				(* Se non ho abilitato il tasteggio in fase di deposito pacco orrizzontale e la missione non prevede deposito orrizzintale do la quota reale*)
				IF TFProgramma_Ciclo_Lastra.DisabilitaDepositoConTasteggio THEN
					TFProgramma_Ciclo_Lastra.Quota_StartLenta_Deposito_Lastra_Z			:= Traiettoria^.PuntoDiApproccioEndPoint.Z;
					TFProgramma_Ciclo_Lastra.Quota_Deposito_Lastra_Z						:= Traiettoria^.EndPoint.Z;
				ELSE // Altrimenti faccio scendere di più l'asse Z in modo da far avvenire il tasteggio.....
					TFProgramma_Ciclo_Lastra.Quota_StartLenta_Deposito_Lastra_Z			:= Traiettoria^.PuntoDiApproccioEndPoint.Z + 10;
					TFProgramma_Ciclo_Lastra.Quota_Deposito_Lastra_Z						:= Traiettoria^.EndPoint.Z - 100;
				END_IF
				
				TFProgramma_Ciclo_Lastra.Quota_Fuori_Ingombro_ConCarico_Z		:= QuotaFuoriIngombro_Z_ConPEZZO;
				TFProgramma_Ciclo_Lastra.Quota_Fuori_Ingombro_SenzaCarico_Z	:= QuotaFuoriIngombro_Z_AVUOTO;
				
				(*J*)
				TFProgramma_Ciclo_Lastra.Quota_Rotazione_Prelievo_Lastra 			:= Traiettoria^.StartPoint.J;
				TFProgramma_Ciclo_Lastra.Quota_Rotazione_Deposito_Lastra 			:= Traiettoria^.EndPoint.J;
				TFProgramma_Ciclo_Lastra();
				IF TFProgramma_Ciclo_Lastra.Inizializzato THEN
					(* Valuto se è abilitata l'interpolazione degli assi *)
					IF NOT AbilitaInterpolazioneAssi^ THEN
						TFWorkFlowCase(ADR(WorkFlow[NumeroWF]),20,WorkflowCase_JMP);	// Case con FB SENZA interpolazione
					ELSE
						TFWorkFlowCase(ADR(WorkFlow[NumeroWF]),30,WorkflowCase_JMP);	// Case con FB CON interpolazione
					END_IF
				END_IF
				
				PaccoPresoXDataLogger := TRUE;
			END_IF;
		(* Case 20 - Chiamata FB del ciclo di lavoro SENZA INTERPOLAZIONE ASSI *)	
		20:	
			TFWorkFlowCase(ADR(WorkFlow[NumeroWF]),30,WorkflowCase_JMP);	// Case con FB CON interpolazione

		
		(* Case 30 - Chiamata FB del ciclo di lavoro CON INTERPOLAZIONE ASSI *)	
		30:	
			IF CmdExe.RapidStopRequest > 0 OR
				TFPalletizerIsModuleError(Modules) THEN
				TFCiclo_Deposito_Lastra.InterrompiCiclo := TRUE;
			ELSE
				TFCiclo_Deposito_Lastra.InterrompiCiclo := FALSE;
			END_IF
			TFCiclo_Deposito_Lastra.Ciclo					:= ADR(Ciclo_Deposito_Lastra);
			TFCiclo_Deposito_Lastra.Programma				:= ADR(TFProgramma_Ciclo_Lastra);
			TFCiclo_Deposito_Lastra.ModuleAX_X 				:= ADR(Modules^.AX_X);
			TFCiclo_Deposito_Lastra.ModuleAX_Y 				:= ADR(Modules^.AX_Y);
			TFCiclo_Deposito_Lastra.ModuleAX_Z 				:= ADR(Modules^.AX_Z);
			TFCiclo_Deposito_Lastra.ModuleAX_J 				:= ADR(Modules^.AX_J);
			TFCiclo_Deposito_Lastra.ModulePinza 		:= ADR(Modules^.Pinza);
			TFCiclo_Deposito_Lastra.StartInterpolazioneAssi 				:= ADR(STARTInterpolazioneASSI^);
			TFCiclo_Deposito_Lastra.AbilitazioneAnticipoDinamicoMovimenti 	:= AbilitaAnticipoDinamico^;
			//TFCiclo_Deposito_Lastra.AbilitaDepositoPaccoOrrizzontaleConTasteggio	:= (AbilitaDepositoPaccoOrrizzonataleConTasteggio^ AND NOT SimulazioneSenzaPalletFalde);
			//TFCiclo_Deposito_Lastra.AbilitaAccostamentoAsseZ						:= AbilitaAccostamentoAsseZ^;
			TFCiclo_Deposito_Lastra.AbilitazioneGlobalePassMode 					:= Traiettoria^.PassModeGlobalEnable;
			TFCiclo_Deposito_Lastra.Abilita_Ciclo_Step								:= AbilitazioCiclo_TEST_STEP;
			
			IF CommandSTEP AND NOT CommandSTEPTRIG THEN
				TFCiclo_Deposito_Lastra.Command_Step	:= TRUE;
				CommandSTEPTRIG := TRUE;
			ELSIF NOT CommandSTEP AND NOT CommandSTEPTRIG THEN
				TFCiclo_Deposito_Lastra.Command_Step	:= FALSE;
				CommandSTEPTRIG := FALSE;
				CommandSTEP := FALSE;
			ELSIF  STEPCicloDONE THEN
				TFCiclo_Deposito_Lastra.Command_Step	:= FALSE;
				CommandSTEP := FALSE;
				CommandSTEPTRIG := FALSE;
			END_IF
			
			TFCiclo_Deposito_Lastra();
			STEPCicloDONE := TFCiclo_Deposito_Lastra.STEPDone;
			
			IF Ciclo_Deposito_Lastra.Stato = TERMINATO THEN
				OUT.StartTilter := TRUE;
				ProductOnGripper := KNOPRODUCT;
				TFWorkFlowCase(ADR(WorkFlow[NumeroWF]),100,WorkflowCase_JMP);
			ELSIF Ciclo_Deposito_Lastra.Stato = INTERROTTO THEN	
				TFWorkFlowCase(ADR(WorkFlow[NumeroWF]),999,WorkflowCase_JMP);	
					
			END_IF

		(* Case 100 *)
		100:WorkFlow[NumeroWF].State := StateWF_END;
			WorkFlow[NumeroWF].Enable := FALSE;
			CommandSTEP := FALSE;
			CommandSTEPTRIG := FALSE;
			ResetComandoRibaltinoEseguito := FALSE;
			AssiInterpolati := FALSE;

		(* Case 999 *)
		(* WorkFlow ERROR *)
		StateWF_ERROR:
			TFWorkFlowError(ADR(WorkFlow[NumeroWF]),ADR(WorkFlowErrorLog[NumeroWF]));
			CmdExe.PhaseStopRequest := 1;
			CmdExe.RapidStopRequest := 1;
			WorkFlow[NumeroWF].Enable := FALSE;
			CommandSTEP := FALSE;
			CommandSTEPTRIG := FALSE;
			AssiInterpolati := FALSE;
		
		ELSE						
			TFWorkFlowError(ADR(WorkFlow[NumeroWF]),ADR(WorkFlowErrorLog[NumeroWF]));
			TFError(ErrNOCMDCASE,ErrNULL,ADR(CmdExe),ADR(State),ADR(Error),ADR(ErrorLog));	
	END_CASE;
END_IF
END_ACTION

ACTION WF09_CicloDepLastraDaWA:
(*-------------------------------------------------------------------------------------------*)
(* WorkFlow 9 -  CICLO DEPOSITO LASTRA PP *)
(*-------------------------------------------------------------------------------------------*)	
NumeroWF := 9;	
IF WorkFlow[NumeroWF].Enable THEN

	IF NOT TFCommandCaseIsEnable(ADR(CmdExe)) THEN RETURN; END_IF
	CASE WorkFlow[NumeroWF].WFCase OF

		(* Case 0 *)
		0:  WorkFlow[NumeroWF].State := StateWF_RUN;
			STEPCicloDONE := FALSE;	
			TFWorkFlowCase(ADR(WorkFlow[NumeroWF]),1,WorkflowCase_INC);
	
		(* Case 1 - Chiamata del FB del ciclo di riposo per Valorizzarne i valori*)
		1:	IF CmdExe.RapidStopRequest > 0  OR
				TFPalletizerIsModuleError(Modules) THEN
				TFWorkFlowCase(ADR(WorkFlow[NumeroWF]),100,WorkflowCase_JMP);
			ELSE

				TFProgramma_Ciclo_Lastra.X_Par := ParametriProgramma_X_CicloLastra;
				TFProgramma_Ciclo_Lastra.Y_Par := ParametriProgramma_Y_CicloLastra;
				TFProgramma_Ciclo_Lastra.Z_Par := ParametriProgramma_Z_CicloLastra;
				TFProgramma_Ciclo_Lastra.J_Par := ParametriProgramma_J_CicloLastra;
				
				(*X*)
				TFProgramma_Ciclo_Lastra.Quota_StartLenta_Prelievo_Lastra_X			:= Traiettoria^.PuntoDiApproccioStartPoint.X;
				TFProgramma_Ciclo_Lastra.Quota_Prelievo_Lastra_X 					:= Traiettoria^.StartPoint.X;
				TFProgramma_Ciclo_Lastra.Quota_StartLenta_Deposito_Lastra_X	 		:= Traiettoria^.PuntoDiApproccioEndPoint.X;	
				TFProgramma_Ciclo_Lastra.Quota_Deposito_Lastra_X 					:= Traiettoria^.EndPoint.X;
				TFProgramma_Ciclo_Lastra.Quota_Fuori_Ingombro_SenzaCarico_X			:= Traiettoria^.EndPoint.X;
				TFProgramma_Ciclo_Lastra.Quota_Fuori_Ingombro_Carico_X				:= Traiettoria^.EndPoint.X;
				
				//*************************
			   	CoordenadaPosGiroPieza_X 											:= WorkArea^[NuPosGuiroPiking].X ;
				TFProgramma_Ciclo_Lastra.Quota_PosGiroPiezaTraCavalleteX			:= CoordenadaPosGiroPieza_X ;
				//*****************************
				
				(*Y*)
				TFProgramma_Ciclo_Lastra.Quota_StartLenta_Prelievo_Lastra_Y         := Traiettoria^.PuntoDiApproccioStartPoint.Y;;
				TFProgramma_Ciclo_Lastra.Quota_Prelievo_Lastra_Y 					:= Traiettoria^.StartPoint.Y;
				TFProgramma_Ciclo_Lastra.Quota_Distacco_Lastra_Y					:= Traiettoria^.PuntoDiPostPosizionamentoStartPoint.Y;
				TFProgramma_Ciclo_Lastra.Quota_StartLenta_Deposito_Lastra_Y			:= Traiettoria^.PuntoDiApproccioEndPoint.Y;
				TFProgramma_Ciclo_Lastra.Quota_Deposito_Lastra_Y 					:= Traiettoria^.EndPoint.Y;
				TFProgramma_Ciclo_Lastra.Quota_Fuori_Ingombro_Y 					:= QuotaFuoriIngombro_Y_ConCARICO;//DEVE ESSERE GUALE A QUELLE DEL CORRIDOIO
				TFProgramma_Ciclo_Lastra.Quota_PasilloCavallete0GradosY             := CoordenadaPasillo0_Y ;
				TFProgramma_Ciclo_Lastra.Quota_PasilloCavallete1800GradosY          := CoordenadaPasillo180_Y ;
			
				(*Z*)
				TFProgramma_Ciclo_Lastra.Quota_StartLenta_Prelievo_Lastra_Z 		:= MAX(Traiettoria^.PuntoDiApproccioStartPoint.Z,AxisPar_Z.MinPosition+1);
				TFProgramma_Ciclo_Lastra.Quota_Prelievo_Lastra_Z 					:= MAX(Traiettoria^.StartPoint.Z,AxisPar_Z.MinPosition+1);
				TFProgramma_Ciclo_Lastra.Quota_StartLenta_Deposito_Lastra_Z			:= Traiettoria^.PuntoDiApproccioEndPoint.Z;
				TFProgramma_Ciclo_Lastra.Quota_Deposito_Lastra_Z					:= MAX(Traiettoria^.EndPoint.Z,AxisPar_Z.MinPosition+1);
				TFProgramma_Ciclo_Lastra.Quota_Fuori_Ingombro_ConCarico_Z			:= QuotaFuoriIngombro_Z_ConPEZZO;
				TFProgramma_Ciclo_Lastra.Quota_Fuori_Ingombro_SenzaCarico_Z			:= QuotaFuoriIngombro_Z_AVUOTO;
				TFProgramma_Ciclo_Lastra.Quota_Distacco_Lastra_Z					:= Traiettoria^.PuntoDiPostPosizionamentoStartPoint.Z;
				TFProgramma_Ciclo_Lastra.Quota_PostScarico							:= Z_Riposo;	
			
				(*J*)
				TFProgramma_Ciclo_Lastra.Quota_Rotazione_Prelievo_Lastra 			:= Traiettoria^.StartPoint.J;
				TFProgramma_Ciclo_Lastra.Quota_Rotazione_Deposito_Lastra 			:= Traiettoria^.EndPoint.J;
				TFProgramma_Ciclo_Lastra.Quota_Rotazione_StartTasteggio_Lastra		:= Traiettoria^.PuntoDiApproccioStartPoint.J;
				TFProgramma_Ciclo_Lastra.Quota_Fuori_Ingombro_J						:= QuotaFuoriIngombro_J_ConCARICO;
				TFProgramma_Ciclo_Lastra.Quota_Rotazione_Sfogliatura 				:= Traiettoria^.StartPoint.J + HMI_GradiSfogliaturaJ;
				TFProgramma_Ciclo_Lastra.Quota_Posicion_Giro_Pinza					:= WorkSpace^.Y / 2 +900;
				TFProgramma_Ciclo_Lastra();
				CommandSTEP := FALSE;
				TFWorkFlowCase(ADR(WorkFlow[NumeroWF]),30,WorkflowCase_JMP);	// Case con FB CON interpolazione
			END_IF;
		(* Case 20 - Chiamata FB del ciclo di lavoro *)	
		20:	
			TFWorkFlowCase(ADR(WorkFlow[NumeroWF]),30,WorkflowCase_JMP);	// Case con FB CON interpolazione

			
		(* Case 30 - Chiamata FB del ciclo di lavoro *)	
		30:	
			IF CmdExe.RapidStopRequest > 0 OR
				TFPalletizerIsModuleError(Modules) OR Error.Code <> 0 THEN
				TFCiclo_Deposito_Lastra.InterrompiCiclo := TRUE;
			ELSE
				TFCiclo_Deposito_Lastra.InterrompiCiclo := FALSE;
			END_IF
			
			EseguitoAllinementoPezziDeposito := FALSE;//Azzeramento per dare la possibilità di allineare le lastre in fase di distacco aspirazione in manuale
			
			TFCiclo_Deposito_Lastra.Ciclo					:= ADR(Ciclo_Deposito_Lastra);
			TFCiclo_Deposito_Lastra.Programma				:= ADR(TFProgramma_Ciclo_Lastra);
			TFCiclo_Deposito_Lastra.ModuleAX_X 				:= ADR(Modules^.AX_X);
			TFCiclo_Deposito_Lastra.ModuleAX_Y 				:= ADR(Modules^.AX_Y);
			TFCiclo_Deposito_Lastra.ModuleAX_Z 				:= ADR(Modules^.AX_Z);
			TFCiclo_Deposito_Lastra.ModuleAX_J 				:= ADR(Modules^.AX_J);
			TFCiclo_Deposito_Lastra.ModulePinza 			:= ADR(Modules^.Pinza);
			TFCiclo_Deposito_Lastra.StartInterpolazioneAssi := ADR(STARTInterpolazioneASSI^);
			TFCiclo_Deposito_Lastra.AbilitazioneAnticipoDinamicoMovimenti 	:= AbilitaAnticipoDinamico^;
			TFCiclo_Deposito_Lastra.AbilitazioneGlobalePassMode 			:= Traiettoria^.PassModeGlobalEnable;
			TFCiclo_Deposito_Lastra.Abilita_Ciclo_Step						:= AbilitazioCiclo_TEST_STEP;
			
			IF CommandSTEP AND NOT CommandSTEPTRIG THEN
				TFCiclo_Deposito_Lastra.Command_Step	:= TRUE;
				CommandSTEPTRIG := TRUE;
			ELSIF NOT CommandSTEP AND NOT CommandSTEPTRIG THEN
				TFCiclo_Deposito_Lastra.Command_Step	:= FALSE;
				CommandSTEPTRIG := FALSE;
				CommandSTEP := FALSE;
			ELSIF  STEPCicloDONE THEN
				TFCiclo_Deposito_Lastra.Command_Step	:= FALSE;
				CommandSTEP := FALSE;
				CommandSTEPTRIG := FALSE;
			END_IF
			
			TFCiclo_Deposito_Lastra();
			STEPCicloDONE := TFCiclo_Deposito_Lastra.STEPDone;
			
			IF TFCiclo_Deposito_Lastra.Ciclo^.Stato = TERMINATO THEN
				ProductOnGripper := KNOPRODUCT;
				TFWorkFlowCase(ADR(WorkFlow[NumeroWF]),100,WorkflowCase_JMP);
			ELSIF TFCiclo_Deposito_Lastra.Errore > 0 THEN
				TFError(TFCiclo_Deposito_Lastra.Errore,ErrNULL,ADR(CmdExe),ADR(State),ADR(Error),ADR(ErrorLog));	
				TFWorkFlowCase(ADR(WorkFlow[NumeroWF]),999,WorkflowCase_JMP);	 
			ELSIF TFCiclo_Deposito_Lastra.Ciclo^.Stato = INTERROTTO THEN	
				TFWorkFlowCase(ADR(WorkFlow[NumeroWF]),999,WorkflowCase_JMP);		
			END_IF

		(* Case 100 *)
		100:WorkFlow[NumeroWF].State := StateWF_END;
			WorkFlow[NumeroWF].Enable := FALSE;
			CommandSTEP := FALSE;
			CommandSTEPTRIG := FALSE;
			AssiInterpolati := FALSE;

		(* Case 999 *)
		(* WorkFlow ERROR *)
		StateWF_ERROR:
			TFWorkFlowError(ADR(WorkFlow[NumeroWF]),ADR(WorkFlowErrorLog[NumeroWF]));
			CmdExe.PhaseStopRequest := 1;
			CmdExe.RapidStopRequest := 1;
			WorkFlow[NumeroWF].Enable := FALSE;
			CommandSTEP := FALSE;
			CommandSTEPTRIG := FALSE;
			AssiInterpolati := FALSE;
		
		ELSE						
			TFWorkFlowError(ADR(WorkFlow[NumeroWF]),ADR(WorkFlowErrorLog[NumeroWF]));
			TFError(ErrNOCMDCASE,ErrNULL,ADR(CmdExe),ADR(State),ADR(Error),ADR(ErrorLog));	
	END_CASE;
END_IF
END_ACTION

ACTION WF10_CicloPelLastra_Depal:
(*-------------------------------------------------------------------------------------------*)
(* WorkFlow 10 -  CICLO PRELIEVO LASTRA DA WA DEPAL*)
(*-------------------------------------------------------------------------------------------*)	
NumeroWF := 10;	
IF WorkFlow[NumeroWF].Enable THEN

	IF NOT TFCommandCaseIsEnable(ADR(CmdExe)) THEN RETURN; END_IF
	CASE WorkFlow[NumeroWF].WFCase OF

		(* Case 0 *)
		0:  WorkFlow[NumeroWF].State := StateWF_RUN;
			STEPCicloDONE := FALSE;	
			OUT.StartTilter := TRUE;
			TFWorkFlowCase(ADR(WorkFlow[NumeroWF]),1,WorkflowCase_INC);
	
		(* Case 1 - Chiamata del FB del ciclo di riposo per Valorizzarne i valori*)
		1:	IF CmdExe.RapidStopRequest > 0 OR
				TFPalletizerIsModuleError(Modules) OR Error.Code <> 0 THEN
				TFWorkFlowCase(ADR(WorkFlow[NumeroWF]),100,WorkflowCase_JMP);
			ELSE
				TFProgramma_Ciclo_Lastra.X_Par := ParametriProgramma_X_CicloLastra;
				TFProgramma_Ciclo_Lastra.Y_Par := ParametriProgramma_Y_CicloLastra;
				TFProgramma_Ciclo_Lastra.Z_Par := ParametriProgramma_Z_CicloLastra;
				TFProgramma_Ciclo_Lastra.J_Par := ParametriProgramma_J_CicloLastra;
				
				(*X*)
				TFProgramma_Ciclo_Lastra.Quota_StartLenta_Prelievo_Lastra_X			:= Traiettoria^.PuntoDiApproccioStartPoint.X;
				TFProgramma_Ciclo_Lastra.Quota_Prelievo_Lastra_X 					:= Traiettoria^.StartPoint.X;
				TFProgramma_Ciclo_Lastra.Quota_StartLenta_Deposito_Lastra_X	 		:= Traiettoria^.PuntoDiApproccioEndPoint.X;	
				TFProgramma_Ciclo_Lastra.Quota_Deposito_Lastra_X 					:= Traiettoria^.EndPoint.X;
				TFProgramma_Ciclo_Lastra.Quota_Fuori_Ingombro_SenzaCarico_X			:= Traiettoria^.EndPoint.X;//STESSA QUOTA DI DEPOSITO X DEPAL UNIVERSAL
				TFProgramma_Ciclo_Lastra.Quota_Fuori_Ingombro_Carico_X				:= Traiettoria^.EndPoint.X;//STESSA QUOTA DI DEPOSITO X DEPAL UNIVERSAL
				
				(*Y*)
				TFProgramma_Ciclo_Lastra.Quota_StartLenta_Prelievo_Lastra_Y         := Traiettoria^.PuntoDiApproccioStartPoint.Y;;
				TFProgramma_Ciclo_Lastra.Quota_Prelievo_Lastra_Y 					:= Traiettoria^.StartPoint.Y;
				TFProgramma_Ciclo_Lastra.Quota_Distacco_Lastra_Y					:= Traiettoria^.PuntoDiPostPosizionamentoStartPoint.Y;
				TFProgramma_Ciclo_Lastra.Quota_StartLenta_Deposito_Lastra_Y			:= Traiettoria^.PuntoDiApproccioEndPoint.Y;
				TFProgramma_Ciclo_Lastra.Quota_Deposito_Lastra_Y 					:= Traiettoria^.EndPoint.Y;
				TFProgramma_Ciclo_Lastra.Quota_Fuori_Ingombro_Y 					:= QuotaFuoriIngombro_Y_AVUOTO;//DEVE ESSERE GUALE A QUELLE DEL CORRIDOIO
				
				(*Z*)
				TFProgramma_Ciclo_Lastra.Quota_StartLenta_Prelievo_Lastra_Z 		:= MAX(Traiettoria^.PuntoDiApproccioStartPoint.Z,AxisPar_Z.MinPosition);
				TFProgramma_Ciclo_Lastra.Quota_Prelievo_Lastra_Z 					:= MAX(Traiettoria^.StartPoint.Z,AxisPar_Z.MinPosition);
				TFProgramma_Ciclo_Lastra.Quota_StartLenta_Deposito_Lastra_Z			:= Traiettoria^.PuntoDiApproccioEndPoint.Z;
				IF HMI_AbilitaDepositoPaccoOrrizzontaleConTasteggio THEN
					TFProgramma_Ciclo_Lastra.Quota_Deposito_Lastra_Z					:= Traiettoria^.EndPoint.Z -100;
				ELSE
					TFProgramma_Ciclo_Lastra.Quota_Deposito_Lastra_Z					:= Traiettoria^.EndPoint.Z;
				END_IF
				TFProgramma_Ciclo_Lastra.Quota_Fuori_Ingombro_ConCarico_Z			:= QuotaFuoriIngombro_Z_ConPEZZO;
				TFProgramma_Ciclo_Lastra.Quota_Fuori_Ingombro_SenzaCarico_Z			:= QuotaFuoriIngombro_Z_AVUOTO;
				TFProgramma_Ciclo_Lastra.Quota_Distacco_Lastra_Z					:= Traiettoria^.PuntoDiPostPosizionamentoStartPoint.Z;
				TFProgramma_Ciclo_Lastra.Quota_PostScarico							:= Z_Riposo;	
			
				(*J*)
				TFProgramma_Ciclo_Lastra.Quota_Rotazione_Prelievo_Lastra 			:= Traiettoria^.StartPoint.J;
				TFProgramma_Ciclo_Lastra.Quota_Rotazione_Deposito_Lastra 			:= Traiettoria^.EndPoint.J;
				TFProgramma_Ciclo_Lastra.Quota_Rotazione_StartTasteggio_Lastra		:= Traiettoria^.StartPoint.J;
				TFProgramma_Ciclo_Lastra.Quota_Fuori_Ingombro_J						:= QuotaFuoriIngombro_J_AVUOTO;
				TFProgramma_Ciclo_Lastra.Quota_Rotazione_Sfogliatura 				:= Traiettoria^.StartPoint.J + HMI_GradiSfogliaturaJ;


				TFProgramma_Ciclo_Lastra();

				(* Valuto se è abilitata l'interpolazione degli assi *)
				IF NOT AbilitaInterpolazioneAssi^ THEN
					TFWorkFlowCase(ADR(WorkFlow[NumeroWF]),20,WorkflowCase_JMP);	// Case con FB SENZA interpolazione
				ELSE
					TFWorkFlowCase(ADR(WorkFlow[NumeroWF]),30,WorkflowCase_JMP);	// Case con FB CON interpolazione
				END_IF
			END_IF;
		(* Case 20 - Chiamata FB del ciclo di lavoro *)	
		20:	
			TFWorkFlowCase(ADR(WorkFlow[NumeroWF]),30,WorkflowCase_JMP);	// Case con FB CON interpolazione

			
		(* Case 30 - Chiamata FB del ciclo di lavoro *)	
		30:	
			IF CmdExe.RapidStopRequest > 0 OR
				TFPalletizerIsModuleError(Modules) OR Error.Code <> 0 THEN
				TFCiclo_Prelievo_Lastra_Depalettizzatore.InterrompiCiclo := TRUE;
			ELSE
				TFCiclo_Prelievo_Lastra_Depalettizzatore.InterrompiCiclo := FALSE;
			END_IF
			//Quota asse J x sfogliatura


			TFCiclo_Prelievo_Lastra.Ciclo					:= ADR(Ciclo_Prelievo_Lastra);
			TFCiclo_Prelievo_Lastra.Programma				:= ADR(TFProgramma_Ciclo_Lastra);
			TFCiclo_Prelievo_Lastra.Modules 				 := Modules;
			TFCiclo_Prelievo_Lastra.StartInterpolazioneAssi := ADR(STARTInterpolazioneASSI^);
			TFCiclo_Prelievo_Lastra.AbilitazioneAnticipoDinamicoMovimenti 	:= AbilitaAnticipoDinamico^;
			TFCiclo_Prelievo_Lastra.AbilitazioneGlobalePassMode 			:= Traiettoria^.PassModeGlobalEnable;
			TFCiclo_Prelievo_Lastra.Abilita_Ciclo_Step						:= AbilitazioCiclo_TEST_STEP;
			TFCiclo_Prelievo_Lastra.PrelievoPezzoOrizzontale				:= TRUE;
			TFCiclo_Prelievo_Lastra.NumeroTentativiPresa					:= HMI_NumeroTentativiPresa;			
		
			IF CommandSTEP AND NOT CommandSTEPTRIG THEN
				TFCiclo_Prelievo_Lastra_Depalettizzatore.Command_Step	:= TRUE;
				CommandSTEPTRIG := TRUE;
			ELSIF NOT CommandSTEP AND NOT CommandSTEPTRIG THEN
				TFCiclo_Prelievo_Lastra_Depalettizzatore.Command_Step	:= FALSE;
				CommandSTEPTRIG := FALSE;
				CommandSTEP := FALSE;
			ELSIF  STEPCicloDONE THEN
				TFCiclo_Prelievo_Lastra_Depalettizzatore.Command_Step	:= FALSE;
				CommandSTEP := FALSE;
				CommandSTEPTRIG := FALSE;
			END_IF
			
			TFCiclo_Prelievo_Lastra_Depalettizzatore();
			STEPCicloDONE := TFCiclo_Prelievo_Lastra_Depalettizzatore.STEPDone;
			
			IF TFCiclo_Prelievo_Lastra_Depalettizzatore.Ciclo^.Stato = TERMINATO THEN
				OUT.StartTilter := TRUE;
				ProductOnGripper := KPRODUCTLOADED;
				TFWorkFlowCase(ADR(WorkFlow[NumeroWF]),100,WorkflowCase_JMP);
			ELSIF TFCiclo_Prelievo_Lastra_Depalettizzatore.Ciclo^.Stato = INTERROTTO OR TFCiclo_Prelievo_Lastra_Depalettizzatore.Errore <> 0 THEN	
				
				IF TFCiclo_Prelievo_Lastra_Depalettizzatore.Errore <> 0 THEN	 
					CmdExe.PhaseStopRequest := 1;
					CmdExe.RapidStopRequest := 1;
					WorkFlow[NumeroWF].Enable := FALSE;
					CommandSTEP := FALSE;
					CommandSTEPTRIG := FALSE;
					AssiInterpolati := FALSE;
					TFCiclo_Prelievo_Lastra_Depalettizzatore.Ciclo^.Stato := INTERROTTO;
					TFCiclo_Prelievo_Lastra_Depalettizzatore.InterrompiCiclo := TRUE;
					TFError(TFCiclo_Prelievo_Lastra_Depalettizzatore.Errore,ErrNULL,ADR(CmdExe),ADR(State),ADR(Error),ADR(ErrorLog));
				ELSE
					TFWorkFlowCase(ADR(WorkFlow[NumeroWF]),999,WorkflowCase_JMP);	
				END_IF	
			END_IF

		(* Case 100 *)
		100:WorkFlow[NumeroWF].State := StateWF_END;
			WorkFlow[NumeroWF].Enable := FALSE;
			CommandSTEP := FALSE;
			CommandSTEPTRIG := FALSE;
			AssiInterpolati := FALSE;

		(* Case 999 *)
		(* WorkFlow ERROR *)
		StateWF_ERROR:
			TFWorkFlowError(ADR(WorkFlow[NumeroWF]),ADR(WorkFlowErrorLog[NumeroWF]));
			CmdExe.PhaseStopRequest := 1;
			CmdExe.RapidStopRequest := 1;
			WorkFlow[NumeroWF].Enable := FALSE;
			CommandSTEP := FALSE;
			CommandSTEPTRIG := FALSE;
			AssiInterpolati := FALSE;
			
		ELSE						
			TFWorkFlowError(ADR(WorkFlow[NumeroWF]),ADR(WorkFlowErrorLog[NumeroWF]));
			TFError(ErrNOCMDCASE,ErrNULL,ADR(CmdExe),ADR(State),ADR(Error),ADR(ErrorLog));	
	END_CASE;
END_IF
END_ACTION

ACTION WF11_CicloDepFalde_Depal:
(*-------------------------------------------------------------------------------------------*)
(* WorkFlow 11 -  CICLO DEPOSITO FALDE DEPAL *)
(*-------------------------------------------------------------------------------------------*)		
NumeroWF := 11;
IF WorkFlow[NumeroWF].Enable THEN

	IF NOT TFCommandCaseIsEnable(ADR(CmdExe)) THEN RETURN; END_IF
	CASE WorkFlow[NumeroWF].WFCase OF

		(* Case 0 *)
		0:  WorkFlow[NumeroWF].State := StateWF_RUN;
			STEPCicloDONE := FALSE;
			OUT.StartTilter := TRUE;
			PaccoPresoXDataLogger := FALSE;
			IF NOT AttivaTimerContaPacchi1Minuto THEN
				AttivaTimerContaPacchi1Minuto := TRUE;
				AttivaTimerContaPacchi5Minuti := TRUE;
				Pacchi1Minuto := Pacchi1Minuto +1;
			ELSIF AttivaTimerContaPacchi1Minuto THEN
				AttivaTimerContaPacchi1Minuto := TRUE;
				Pacchi1Minuto := Pacchi1Minuto +1;
			END_IF	
			
			TFWorkFlowCase(ADR(WorkFlow[NumeroWF]),1,WorkflowCase_INC);
	
				(* Case 1 - Chiamata del FB del ciclo di riposo per Valorizzarne i valori*)
		1:	IF CmdExe.RapidStopRequest > 0 OR
				TFPalletizerIsModuleError(Modules) OR Error.Code <> 0 THEN
				TFWorkFlowCase(ADR(WorkFlow[NumeroWF]),100,WorkflowCase_JMP);
			ELSE
				TFProgramma_Ciclo_Falda.X_Par := ParametriProgramma_X_CicloFalda;
				TFProgramma_Ciclo_Falda.Y_Par := ParametriProgramma_Y_CicloFalda;
				TFProgramma_Ciclo_Falda.Z_Par := ParametriProgramma_Z_CicloFalda;
				TFProgramma_Ciclo_Falda.J_Par := ParametriProgramma_J_CicloFalda;
				
				(*X*)
				//TFProgramma_Ciclo_Falda.Quota_Prelievo_Falda_X 					:= Traiettoria^.StartPoint.X;
				//TFProgramma_Ciclo_Falda.Quota_Deposito_Falda_SuCatastaPallet_X 	:= Traiettoria^.EndPoint.X;
				TFProgramma_Ciclo_Falda.Quota_Deposito_Falda_SuPiazzola_X	 	:= Traiettoria^.EndPointSecondario.X;	
				//TFProgramma_Ciclo_Falda.Quota_Deposito_Falda_SuPiazzola_X	 	:= Traiettoria^.EndPointSecondario.X;	
				(*Y*)
				//TFProgramma_Ciclo_Falda.Quota_Prelievo_Falda_Y 					:= Traiettoria^.StartPoint.Y;
				TFProgramma_Ciclo_Falda.Quota_Deposito_Falda_SuCatastaPallet_Y 	:= Traiettoria^.EndPointSecondario.Y;
				TFProgramma_Ciclo_Falda.Quota_Deposito_Falda_SuPiazzola_Y		:= Traiettoria^.EndPointSecondario.Y;
				TFProgramma_Ciclo_Falda.Quota_Fuori_Ingombro_Y 					:= QuotaFuoriIngombro_Y_ConCARICO;

				(*Z*)
				//TFProgramma_Ciclo_Falda.Quota_StartLenta_Prelievo_Falda_Z 					:= Traiettoria^.PuntoDiApproccioStartPoint.Z;
				//TFProgramma_Ciclo_Falda.Quota_Prelievo_Falda_Z 								:= Traiettoria^.StartPoint.Z;
				TFProgramma_Ciclo_Falda.Quota_StartLenta_Deposito_Falda_SuPiazzola_Z 		:= Traiettoria^.PuntoDiApproccioSecondarioEndPoint.Z;
				TFProgramma_Ciclo_Falda.Quota_Deposito_Falda_SuPiazzola_Z					:= Traiettoria^.EndPointSecondario.Z;
				TFProgramma_Ciclo_Falda.Quota_StartLenta_Deposito_Falda_SuCatastaPallet_Z	:= Traiettoria^.PuntoDiApproccioSecondarioEndPoint.Z;
				TFProgramma_Ciclo_Falda.Quota_Deposito_Falda_SuCatastaPallet_Z				:= Traiettoria^.EndPointSecondario.Z;
				TFProgramma_Ciclo_Falda.QUota_Fuori_Ingombro_Falda_Z 						:= QuotaFuoriIngombro_Z_ConPEZZO;
				//TFProgramma_Ciclo_Falda.Quota_Attesa_Caduta_Falda_Z							:= Modules^.AX_Z.Ax^.Status.ActPosition + OffsetCadutaFalda;//Quota_Attesa_Caduta_Falda_Z;
					
				(*J*)
				//TFProgramma_Ciclo_Falda.Quota_Rotazione_Prelievo_Falda 			:= Traiettoria^.StartPoint.J;
				TFProgramma_Ciclo_Falda.Quota_Rotazione_Deposito_Falda 			:= 90;//Traiettoria^.EndPoint.J;
				TFProgramma_Ciclo_Falda();
				(* Valuto se è abilitata l'interpolazione degli assi *)
				IF NOT AbilitaInterpolazioneAssi^ THEN
					TFWorkFlowCase(ADR(WorkFlow[NumeroWF]),20,WorkflowCase_JMP);	// Case con FB SENZA interpolazione
				ELSE
					TFWorkFlowCase(ADR(WorkFlow[NumeroWF]),30,WorkflowCase_JMP);	// Case con FB CON interpolazione
				END_IF
			END_IF;
		(* Case 20 - Chiamata FB del ciclo di lavoro *)	
		20:	
			TFWorkFlowCase(ADR(WorkFlow[NumeroWF]),30,WorkflowCase_JMP);	// Case con FB CON interpolazione

			
		(* Case 30 - Chiamata FB del ciclo di lavoro *)	
		30:	
			IF CmdExe.RapidStopRequest > 0 OR
				TFPalletizerIsModuleError(Modules) OR Error.Code <> 0 THEN
				TFCiclo_Deposito_Falda_Depalettizzatore.InterrompiCiclo := TRUE;
			ELSE
				TFCiclo_Deposito_Falda_Depalettizzatore.InterrompiCiclo := FALSE;
			END_IF
			TFCiclo_Deposito_Falda_Depalettizzatore.Ciclo					:= ADR(Ciclo_Deposito_Falda_Depal);
			TFCiclo_Deposito_Falda_Depalettizzatore.Programma				:= ADR(TFProgramma_Ciclo_Falda);
			TFCiclo_Deposito_Falda_Depalettizzatore.ModuleAX_X 				:= ADR(Modules^.AX_X);
			TFCiclo_Deposito_Falda_Depalettizzatore.ModuleAX_Y 				:= ADR(Modules^.AX_Y);
			TFCiclo_Deposito_Falda_Depalettizzatore.ModuleAX_Z 				:= ADR(Modules^.AX_Z);
			TFCiclo_Deposito_Falda_Depalettizzatore.ModuleAX_J 				:= ADR(Modules^.AX_J);
			TFCiclo_Deposito_Falda_Depalettizzatore.ModulePinza 			:= ADR(Modules^.Pinza);
			TFCiclo_Deposito_Falda_Depalettizzatore.StartInterpolazioneAssi 			:= ADR(STARTInterpolazioneASSI^);
			TFCiclo_Deposito_Falda_Depalettizzatore.AbilitazioneGlobalePassMode 		:= Traiettoria^.PassModeGlobalEnable;
			TFCiclo_Deposito_Falda_Depalettizzatore.Abilita_Ciclo_Step		:= AbilitazioCiclo_TEST_STEP;
			(* Set della tipologia di deposito *)
		//	IF Workarea^[Mission^.PPlace].Typology = TYPOLOGY_STACK THEN 
			//	TFCiclo_Deposito_Falda_Depalettizzatore.TipoDiDeposito		:= DEPOSITO_FALDA_SU_CATASTA;
			//ELSIF Workarea^[Mission^.PPlace].Typology = TYPOLOGY_PALLET THEN
				TFCiclo_Deposito_Falda_Depalettizzatore.TipoDiDeposito		:= DEPOSITO_FALDA_SU_PIAZZOLA;
			//ELSE
				//; //non dovrebbe mai accadere
			//END_IF
			
			IF CommandSTEP AND NOT CommandSTEPTRIG THEN
				TFCiclo_Deposito_Falda_Depalettizzatore.Command_Step	:= TRUE;
				CommandSTEPTRIG := TRUE;
			ELSIF NOT CommandSTEP AND NOT CommandSTEPTRIG THEN
				TFCiclo_Deposito_Falda_Depalettizzatore.Command_Step	:= FALSE;
				CommandSTEPTRIG := FALSE;
				CommandSTEP := FALSE;
			ELSIF  STEPCicloDONE THEN
				TFCiclo_Deposito_Falda_Depalettizzatore.Command_Step	:= FALSE;
				CommandSTEP := FALSE;
				CommandSTEPTRIG := FALSE;
			END_IF
			
			TFCiclo_Deposito_Falda_Depalettizzatore();
			STEPCicloDONE := TFCiclo_Deposito_Falda_Depalettizzatore.STEPDone;
			
			IF Ciclo_Deposito_Falda_Depal.Stato = TERMINATO THEN
				OUT.StartTilter := TRUE;
				ProductOnGripper := KNOPRODUCT;
				TFWorkFlowCase(ADR(WorkFlow[NumeroWF]),100,WorkflowCase_JMP);
			ELSIF Ciclo_Deposito_Falda_Depal.Stato = INTERROTTO THEN	
				TFWorkFlowCase(ADR(WorkFlow[NumeroWF]),999,WorkflowCase_JMP);		
			END_IF

		(* Case 100 *)
		100:WorkFlow[NumeroWF].State := StateWF_END;
			WorkFlow[NumeroWF].Enable := FALSE;
			CommandSTEP := FALSE;
			CommandSTEPTRIG := FALSE;
			TFWorkFlowCase(ADR(WorkFlow[NumeroWF]),0,WorkflowCase_JMP);
			AssiInterpolati := FALSE;

		(* Case 999 *)
		(* WorkFlow ERROR *)
		StateWF_ERROR:
			TFWorkFlowError(ADR(WorkFlow[NumeroWF]),ADR(WorkFlowErrorLog[NumeroWF]));
			CmdExe.PhaseStopRequest := 1;
			CmdExe.RapidStopRequest := 1;
			WorkFlow[NumeroWF].Enable := FALSE;
			CommandSTEP := FALSE;
			CommandSTEPTRIG := FALSE;
			AssiInterpolati := FALSE;
		
		ELSE						
			TFWorkFlowError(ADR(WorkFlow[NumeroWF]),ADR(WorkFlowErrorLog[NumeroWF]));
			TFError(ErrNOCMDCASE,ErrNULL,ADR(CmdExe),ADR(State),ADR(Error),ADR(ErrorLog));	
	END_CASE;
END_IF
END_ACTION

ACTION WF12_CicloDepLastra_Depal:
(*-------------------------------------------------------------------------------------------*)
(* WorkFlow 12 -  CICLO DEPOSITO LASTRA DEPAL *)
(*-------------------------------------------------------------------------------------------*)		
NumeroWF := 12;
IF WorkFlow[NumeroWF].Enable THEN

	IF NOT TFCommandCaseIsEnable(ADR(CmdExe)) THEN RETURN; END_IF
	CASE WorkFlow[NumeroWF].WFCase OF

		(* Case 0 *)
		0:  WorkFlow[NumeroWF].State := StateWF_RUN;
			STEPCicloDONE := FALSE;
			OUT.StartTilter := TRUE;
			PaccoPresoXDataLogger := FALSE;
			IF NOT AttivaTimerContaPacchi1Minuto THEN
				AttivaTimerContaPacchi1Minuto := TRUE;
				AttivaTimerContaPacchi5Minuti := TRUE;
				Pacchi1Minuto := Pacchi1Minuto +1;
			ELSIF AttivaTimerContaPacchi1Minuto THEN
				AttivaTimerContaPacchi1Minuto := TRUE;
				Pacchi1Minuto := Pacchi1Minuto +1;
			END_IF	
			
			TFWorkFlowCase(ADR(WorkFlow[NumeroWF]),1,WorkflowCase_INC);
	
		(* Case 1 - Chiamata del FB del ciclo di riposo per Valorizzarne i valori*)
		1:	IF CmdExe.RapidStopRequest > 0 OR
				TFPalletizerIsModuleError(Modules) OR Error.Code <> 0 THEN
				TFWorkFlowCase(ADR(WorkFlow[NumeroWF]),100,WorkflowCase_JMP);
			ELSE
				TFProgramma_Ciclo_Lastra.X_Par := ParametriProgramma_X_CicloLastra;
				TFProgramma_Ciclo_Lastra.Y_Par := ParametriProgramma_Y_CicloLastra;
				TFProgramma_Ciclo_Lastra.Z_Par := ParametriProgramma_Z_CicloLastra;
				TFProgramma_Ciclo_Lastra.J_Par := ParametriProgramma_J_CicloLastra;
				
				(*X*)
				TFProgramma_Ciclo_Lastra.Quota_StartLenta_Prelievo_Lastra_X			:= Traiettoria^.PuntoDiApproccioStartPoint.X;
				TFProgramma_Ciclo_Lastra.Quota_Prelievo_Lastra_X 					:= Traiettoria^.StartPoint.X;
				TFProgramma_Ciclo_Lastra.Quota_StartLenta_Deposito_Lastra_X	 		:= Traiettoria^.PuntoDiApproccioEndPoint.X;	
				TFProgramma_Ciclo_Lastra.Quota_Deposito_Lastra_X 					:= Traiettoria^.EndPoint.X;
				TFProgramma_Ciclo_Lastra.Quota_Fuori_Ingombro_SenzaCarico_X			:= Traiettoria^.EndPoint.X;//STESSA QUOTA DI DEPOSITO X DEPAL UNIVERSAL
				TFProgramma_Ciclo_Lastra.Quota_Fuori_Ingombro_Carico_X				:= Traiettoria^.EndPoint.X;//STESSA QUOTA DI DEPOSITO X DEPAL UNIVERSAL
				
				(*Y*)
				TFProgramma_Ciclo_Lastra.Quota_StartLenta_Prelievo_Lastra_Y         := Traiettoria^.PuntoDiApproccioStartPoint.Y;;
				TFProgramma_Ciclo_Lastra.Quota_Prelievo_Lastra_Y 					:= Traiettoria^.StartPoint.Y;
				TFProgramma_Ciclo_Lastra.Quota_Distacco_Lastra_Y					:= Traiettoria^.PuntoDiPostPosizionamentoStartPoint.Y;
				TFProgramma_Ciclo_Lastra.Quota_StartLenta_Deposito_Lastra_Y			:= Traiettoria^.PuntoDiApproccioEndPoint.Y;
				TFProgramma_Ciclo_Lastra.Quota_Deposito_Lastra_Y 					:= Traiettoria^.EndPoint.Y;
				TFProgramma_Ciclo_Lastra.Quota_Fuori_Ingombro_Y 					:= QuotaFuoriIngombro_Y_ConCARICO;//DEVE ESSERE GUALE A QUELLE DEL CORRIDOIO
				
				(*Z*)
				TFProgramma_Ciclo_Lastra.Quota_StartLenta_Prelievo_Lastra_Z 		:= Traiettoria^.PuntoDiApproccioStartPoint.Z;
				TFProgramma_Ciclo_Lastra.Quota_Prelievo_Lastra_Z 					:= Traiettoria^.StartPoint.Z;
				TFProgramma_Ciclo_Lastra.Quota_StartLenta_Deposito_Lastra_Z			:= Traiettoria^.PuntoDiApproccioEndPoint.Z;// + PickPlaceParameters^.ZPlaceApproach;//OffsetSicurezza.Z.Carico;
				TFProgramma_Ciclo_Lastra.Quota_Deposito_Lastra_Z					:= Traiettoria^.EndPoint.Z;
				TFProgramma_Ciclo_Lastra.Quota_Fuori_Ingombro_ConCarico_Z			:= QuotaFuoriIngombro_Z_ConPEZZO;
				TFProgramma_Ciclo_Lastra.Quota_Fuori_Ingombro_SenzaCarico_Z			:= QuotaFuoriIngombro_Z_AVUOTO;
				TFProgramma_Ciclo_Lastra.Quota_Distacco_Lastra_Z					:= Traiettoria^.PuntoDiPostPosizionamentoStartPoint.Z;
				TFProgramma_Ciclo_Lastra.Quota_PostScarico							:= Traiettoria^.EndPoint.Z + 30; //Z_Riposo;

				(*J*)
				TFProgramma_Ciclo_Lastra.Quota_Rotazione_Prelievo_Lastra 			:= Traiettoria^.StartPoint.J;
				TFProgramma_Ciclo_Lastra.Quota_Rotazione_Deposito_Lastra 			:= Traiettoria^.EndPoint.J;
				TFProgramma_Ciclo_Lastra.Quota_Rotazione_StartTasteggio_Lastra		:= Traiettoria^.PuntoDiApproccioStartPoint.J;
				TFProgramma_Ciclo_Lastra.Quota_Fuori_Ingombro_J						:= QuotaFuoriIngombro_J_ConCARICO;
				TFProgramma_Ciclo_Lastra();

				IF TFProgramma_Ciclo_Lastra.Inizializzato THEN
					(* Valuto se è abilitata l'interpolazione degli assi *)
					IF NOT AbilitaInterpolazioneAssi^ THEN
						TFWorkFlowCase(ADR(WorkFlow[NumeroWF]),20,WorkflowCase_JMP);	// Case con FB SENZA interpolazione
					ELSE
						TFWorkFlowCase(ADR(WorkFlow[NumeroWF]),30,WorkflowCase_JMP);	// Case con FB CON interpolazione
					END_IF
				END_IF
				
				PaccoPresoXDataLogger := FALSE;
			END_IF;
		(* Case 20 - Chiamata FB del ciclo di lavoro SENZA INTERPOLAZIONE ASSI *)	
		20:	
			TFWorkFlowCase(ADR(WorkFlow[NumeroWF]),30,WorkflowCase_JMP);	// Case con FB CON interpolazione

		
		(* Case 30 - Chiamata FB del ciclo di lavoro CON INTERPOLAZIONE ASSI *)	
		30:	
			IF CmdExe.RapidStopRequest > 0 OR
				TFPalletizerIsModuleError(Modules) OR Error.Code <> 0 OR 
				(CmdExe.PhaseStopRequest > 0 AND Ciclo_Deposito_Lastra_Depal.Passo = 56 AND NOT OkDepositoDaLinea) THEN
				TFCiclo_Deposito_Lastra_Depalettizzatore.InterrompiCiclo := TRUE;
			ELSE
				TFCiclo_Deposito_Lastra_Depalettizzatore.InterrompiCiclo := FALSE;
			END_IF
			TFCiclo_Deposito_Lastra_Depalettizzatore.Ciclo					:= ADR(Ciclo_Deposito_Lastra_Depal);
			TFCiclo_Deposito_Lastra_Depalettizzatore.Programma				:= ADR(TFProgramma_Ciclo_Lastra);
			TFCiclo_Deposito_Lastra_Depalettizzatore.ModuleAX_X 				:= ADR(Modules^.AX_X);
			TFCiclo_Deposito_Lastra_Depalettizzatore.ModuleAX_Y 				:= ADR(Modules^.AX_Y);
			TFCiclo_Deposito_Lastra_Depalettizzatore.ModuleAX_Z 				:= ADR(Modules^.AX_Z);
			TFCiclo_Deposito_Lastra_Depalettizzatore.ModuleAX_J 				:= ADR(Modules^.AX_J);
			TFCiclo_Deposito_Lastra_Depalettizzatore.ModulePinza 		:= ADR(Modules^.Pinza);
			TFCiclo_Deposito_Lastra_Depalettizzatore.StartInterpolazioneAssi 				:= ADR(STARTInterpolazioneASSI^);
			TFCiclo_Deposito_Lastra_Depalettizzatore.AbilitazioneAnticipoDinamicoMovimenti 	:= AbilitaAnticipoDinamico^;
			TFCiclo_Deposito_Lastra_Depalettizzatore.AbilitazioneGlobalePassMode 					:= Traiettoria^.PassModeGlobalEnable;
			TFCiclo_Deposito_Lastra_Depalettizzatore.Abilita_Ciclo_Step								:= AbilitazioCiclo_TEST_STEP;
			//TFCiclo_Deposito_Lastra_Depalettizzatore.MaterialeDepositatoSuLinea	=> MaterialeDepositatoSuLinea;	
	
			IF CommandSTEP AND NOT CommandSTEPTRIG THEN
				TFCiclo_Deposito_Lastra_Depalettizzatore.Command_Step	:= TRUE;
				CommandSTEPTRIG := TRUE;
			ELSIF NOT CommandSTEP AND NOT CommandSTEPTRIG THEN
				TFCiclo_Deposito_Lastra_Depalettizzatore.Command_Step	:= FALSE;
				CommandSTEPTRIG := FALSE;
				CommandSTEP := FALSE;
			ELSIF  STEPCicloDONE THEN
				TFCiclo_Deposito_Lastra_Depalettizzatore.Command_Step	:= FALSE;
				CommandSTEP := FALSE;
				CommandSTEPTRIG := FALSE;
			END_IF
			
			TFCiclo_Deposito_Lastra_Depalettizzatore();
			STEPCicloDONE := TFCiclo_Deposito_Lastra_Depalettizzatore.STEPDone;
			
			IF Ciclo_Deposito_Lastra_Depal.Stato = TERMINATO THEN
				OUT.StartTilter := TRUE;
				ProductOnGripper := KNOPRODUCT;
				TFWorkFlowCase(ADR(WorkFlow[NumeroWF]),100,WorkflowCase_JMP);
			ELSIF (Ciclo_Deposito_Lastra_Depal.Stato = INTERROTTO AND (CmdExe.RapidStopRequest > 0 OR CmdExe.PhaseStopRequest > 0) AND Ciclo_Deposito_Lastra_Depal.Passo = 56 AND NOT OkDepositoDaLinea) THEN
				TFWorkFlowCase(ADR(WorkFlow[NumeroWF]),100,WorkflowCase_JMP);
			ELSIF Ciclo_Deposito_Lastra_Depal.Stato = INTERROTTO THEN	
				TFWorkFlowCase(ADR(WorkFlow[NumeroWF]),999,WorkflowCase_JMP);	
			END_IF

		(* Case 100 *)
		100:WorkFlow[NumeroWF].State := StateWF_END;
			WorkFlow[NumeroWF].Enable := FALSE;
			CommandSTEP := FALSE;
			CommandSTEPTRIG := FALSE;
			ResetComandoRibaltinoEseguito := FALSE;
			AssiInterpolati := FALSE;

		(* Case 999 *)
		(* WorkFlow ERROR *)
		StateWF_ERROR:
			TFWorkFlowError(ADR(WorkFlow[NumeroWF]),ADR(WorkFlowErrorLog[NumeroWF]));
			CmdExe.PhaseStopRequest := 1;
			CmdExe.RapidStopRequest := 1;
			WorkFlow[NumeroWF].Enable := FALSE;
			CommandSTEP := FALSE;
			CommandSTEPTRIG := FALSE;
			AssiInterpolati := FALSE;
		
		ELSE						
			TFWorkFlowError(ADR(WorkFlow[NumeroWF]),ADR(WorkFlowErrorLog[NumeroWF]));
			TFError(ErrNOCMDCASE,ErrNULL,ADR(CmdExe),ADR(State),ADR(Error),ADR(ErrorLog));	
	END_CASE;
END_IF
END_ACTION

END_FUNCTION_BLOCK

// ---- POUs/TFPalletizerDataTF/NON_USATE/TFPalletizerWorkAreaManagerTF.TcPOU
FUNCTION_BLOCK TFPalletizerWorkAreaManagerTF
VAR_INPUT
	Cfg : Config;
	WorkArea : POINTER TO ARRAY [1..MAXAREA] OF TFMachinePalletizer_WorkArea;
	WorkAreaState : POINTER TO ARRAY [1..MAXAREA] OF TFMachinePalletizer_WorkAreaState;
	WorkAreaOffset : POINTER TO ARRAY [1..MAXAREA] OF TFMachinePalletizer_WorkAreaOffset;
	PX_WorkArea : ARRAY [1..MAXAREA] OF BOOL;
	WorkPickPoint : POINTER TO ARRAY [1..MAXPICKPOINT] OF TFMachinePalletizer_WorkPickPoint;
	WorkPickPointOffset : POINTER TO ARRAY [1..MAXPICKPOINT] OF TFMachinePalletizer_WorkPPOffset;
	WorkPickPointState : POINTER TO ARRAY [1..MAXPICKPOINT] OF TFMachinePalletizer_WorkPickPointState;
	Forming : POINTER TO ARRAY [1..MAXFORMING] OF TFMachinePalletizer_Forming;
	Pallet : POINTER TO ARRAY [1..MAXPALLET] OF TFMachinePalletizer_Pallet;
	Layer : POINTER TO ARRAY [1..MAXLAYER] OF TFMachinePalletizer_Layer;
	Mission : POINTER TO TFMachinePalletizer_Mission;
	PickPlaceParameters	: POINTER TO TFMachinePalletizer_ParametersFromHMI;
	ExternalWaitPositionRequest : BOOL;
	ProgressiveNrWA : POINTER TO UDINT;
	UsedCode : POINTER TO ARRAY [1..MAXFORMINGCODE] OF INT;
	TCPParameter : POINTER TO TFModulePalletizerRobot_TCPPar;
	TilterPack : POINTER TO ARRAY [1..MAXHANDLINGSTACK] OF TFHandlingPack;
	PreviousPWA : POINTER TO INT;
	RestoreCWA : POINTER TO BOOL;
	PreviousStackWA : POINTER TO INT;
	WorkAreaManager : POINTER TO TFWorkAreaManager;
	ModuleAX_X : POINTER TO TFModulePalletizer_Ax;
	ModuleAX_Y : POINTER TO TFModulePalletizer_Ax;
	ModuleAX_Z : POINTER TO TFModulePalletizer_Ax;
	ModuleAX_J : POINTER TO TFModulePalletizer_Ax;
	ModuleAX_K : POINTER TO TFModulePalletizer_Ax;
	
	WorkAreaZone : POINTER TO TFMachinePalletizer_WorkAreaZone;	// Struttura delle zone di lavoro
	//HandlingPackTable : POINTER TO TFHandlingPackTable;			// Tabella contenente i pacchi sui trasporti
	ArrayPacchi : POINTER TO DUT_ArrayPacchi; 					//Array contenente i pacchi sui trasporti				
	GestioneAZoneAbilitata : POINTER TO BOOL;					// Abilitazione della gestione a zone
	HandlingRun : BOOL;											//Traspoti in Automatico
	RichiestaStartRibaltino : BOOL;
	AbilitaForzaturaStatoDaRiposoAPrelievo : POINTER TO BOOL;			// Abilita il cambio al volo della missione dal ciclo di riposo al ciclo di prelievo
	AbilitaDisposizionePalletContinua : POINTER TO BOOL;				// Abilitazione del deposito dei pallet ogni qualvolta il carico imposto dalla line a soddisfi determinato requisiti
	AbilitaDepositoPaccoOrrizzonataleConTasteggio : POINTER TO BOOL; 	// Abilitazione per il deposito del pacco con tasteggio del pacco orrizzontale
	AbilitaAssegnazioneCodicePiazzoleConPaccoSuRibaltino : BOOL := TRUE; // Abilitazione della gestione del codice in modo opportunistico rispettando le zone
	AbilitaOffsetInUscitaTasteggioPrelievoPallet : POINTER TO BOOL; 	// Abilitazione dell'offset in uscita dei tastatori in prelievo pallet con tasteggio
END_VAR
VAR_OUTPUT
	InWaitPosition : BOOL;
	DepositoPaccoInLenta : BOOL;					// TRUE: Il deposito del pacco deve avvenire in lenta
	ForzaPrelievoPaccoDuranteCicloDiRiposo : BOOL; // Indica che il ciclo sta facendo un salto: Da ciclo di riposo -> A ciclo di prelievo 
	Errore : uint; //Codice di errore del WorkAreaManager
END_VAR
VAR
	TimerPositionMission : REAL;
	TimerDepositoContinuoPallet : REAL;
	//TimerAttesaAssegnazioneCodice : REAL;
	CurrentWorkArea : INT;
	cwa : INT;
	pwa : INT;
	wa : INT;
	pf : INT;
	pp : INT;
	fcode : INT;
	pcode : INT;
	pcodeUnassigned : INT;
	ppick : INT;
	lpick : INT;
	jp : INT;
	torque : REAL;
	kpick : REAL;
	XPick : REAL;
	YPick : REAL;
	ZPick : REAL;
	JPick : REAL;
	HalfPackDim : REAL;
	vo : INT;
	UnloadOnWADisabled : BOOL;
	EnableCode : ARRAY [1..MAXFORMINGCODE*MAXFORMING] OF INT;
	NFreeWA : INT;
	WAPointer : ARRAY [1..MAXAREA] OF TFMachinePalletizer_WorkAreaSort;
	ZOffsetPick : REAL;
	ZOffsetPlace : REAL;
	DifferenceRealNominalDimensionZ :REAL;
	WaitPositionRequest : BOOL;
	WaitPositionRequestTRIG : BOOL;
	BypassTEST : BOOL;							// ByPASS per il conteggio dei pacchi durante le simulazioni
	PaccoSuRibaltinoDuranteCicloRiposo : BOOL; // Indica che il pacco è pronto durante sul ribaltino mentre il braccio sta andando sul punto di riposo
	CicloDiRiposoNecessario : BOOL;		// Forzatura del ciclo di riposo da parte del WAManager
	OKDepositoPalletContinuo : BOOL;	// Indica che la linea è in uno stato da consentire il deposito continuo dei pallet
	NPacchiPresentiSuLinea : UINT;		// Indica il numero dei pacchi presenti sulla linea
	NUltimiTrasportiOccupati : UINT;	// Indica il numero di trasporti occupati a partire dal ribaltino
	HandlingOKPrelievoPacco : BOOL; 	// Indica che il Ribaltino è pronto a consegnare il pacco
	ConsentiDepositoPaccoSuWA : BOOL; 	// Indica il Pacco può essere depositato sulla WorkArea
	RibaltinoOKPerDepositoContinuo : BOOL; 	// Viene settato quando il ribaltino non è in fase di consegna pacco alla pinza da un certo Tempo (TimerDepositoContinuoPallet)
	NumeroRibaltinoOccupatoConCodicePiazzola : INT; // Indica il ribaltino Avente un pacco con il codice uguale a quello della WA in esame
	ComandoRibaltino : INT;							// Indica il comando Imposto al ribaltino
	ConsentiMovimentoRibaltino : BOOL;				// Indica che il ribaltino può compiere i vari movimenti per posizionare il pacco in prelievo
	AbilitaComandiAnticipatiRibaltino : BOOL;		// Abilitazione dell'anticipo dei comandi del ribaltino ( TRUE:il ribaltino si posiziona in qualsiasi posizione della pinza,FALSE: il ribaltino si posiziona solo quando la pinza è sul punto di prelievo) 
	DisabilitaApproccioPacciOrrizzontali : BOOL := TRUE; // Abilitazione dell'approccio per i pacchi orrizzontali, in questo modo il ciclo è più rapido
	QuotaFittizziaPerTasteggioDepPacchi : REAL := 200; //Quota fittizzia per consentire il tasteggio durante il deposito dei pacci orrizzontali
	UltimaPoastazioneDiAssegnazione : INT;				// Variabile per Debug Interno
	UltimoComando : INT;								// Variabile per Debug Interno
	UltimoStatoCMDRibaltino : INT;						// Variabile per Debug Interno
	WAconCodiceWPPPresente : BOOL;						// Indica che esiste almento una WA in lavorazione con il codice del pacco presente sul ribaltino in questione
	FormaturaAttivaMista : BOOL;						// Indica che la formatura attiva è di tipo Misto (FALSE:utilizzata per anticipare ulteriormente il ribaltino,TRUE:si aspetta che sia terminato il deposito del pacco in corso prima di comandare il ribaltino)
	PalletDepositatiSenzaCodicePresenti : BOOL;			// Indica che sono presenti dei pallet depositati con codice 0 ( Per assegnazione codice in modalità opportunistica(In base al codice sul ribaltino))
	CodiceValidoPerWA : BOOL;							// Indica che il codice del pacco sul ribaltino è presente nella formatura attiva nella WA considerata

	SimulazioneSenzaPallet : BOOL; //Variabile per simulare in officina senza pacco e pallet
	PalletPrelevatiXSimulazione : INT;
	PalletPrelevatiSimulazioneMAX : INT:= 5;
	
	ComandoPickPoint : ARRAY[1..10] OF INT;
	StatoPickPoint : ARRAY[1..10] OF INT;
	cmd : INT :=1;
	FormatureMultipleAttive : BOOL;	//Indica che ci sono più formature Diverse ABILITATE
	UltimaWAAssegnazionePacco : int; //debug
	WAAssegnazionePaccoNONok: BOOL;//debug
	wapick : INT;
	i : uint;
END_VAR

//SimulazioneSenzaPallet := TRUE;


//TFPalletizerWorkAreaManagerTF := FALSE;
(* Chiamata del timer per andare alla posizione di riposo *)
TFTimerCall(ADR(TimerPositionMission),Cfg.TimeBase);
TFTimerCall(ADR(TimerDepositoContinuoPallet),Cfg.TimeBase);
//TFTimerCall(ADR(TimerAttesaAssegnazioneCodice),Cfg.TimeBase);
(* Inizializzazione del WAM *)
Errore := 0;//Azzeramento errore;
IF WorkAreaManager^.State = -1 THEN
	WorkAreaManager^.State := WAMANAGER_NOP;
	ExternalWaitPositionRequest := TRUE;
END_IF

(* Set quota per il tasteggio per deposito pacco orrizzontale *)
QuotaFittizziaPerTasteggioDepPacchi := 200;

(* Set codici abilitati *)
//EnableCode := TFGetEnableCode(Forming);
(*****************************************************************************************************************************)
(* Gestione dello stop in fase -> Si aspetta che si abbia finito la missione e si porta il Braccio nella posizione di riposo *)
(*****************************************************************************************************************************)
(* Set della condizione di posizione di riposo Wait Position *)
InWaitPosition := TFPalletizerInPosizioneRiposo(ModuleAX_X,ModuleAX_Y,ModuleAX_Z,ModuleAX_J,ModuleAX_K,Mission);
IF Mission^.State <> MISSION_STATE_NOP THEN
	TFTimerSet(ADR(TimerPositionMission),200,TRUE);
END_IF
IF ((ExternalWaitPositionRequest AND WorkAreaManager^.State = WAMANAGER_NOP) OR TFTimerDone(ADR(TimerPositionMission))) AND NOT InWaitPosition THEN
	WaitPositionRequestTRIG := TRUE;
END_IF
IF 	WaitPositionRequestTRIG THEN
	WaitPositionRequest := TRUE;
END_IF
IF WaitPositionRequestTRIG AND WaitPositionRequest AND (InWaitPosition AND WorkAreaManager^.State = WAMANAGER_NOP) THEN
	WaitPositionRequest := FALSE;
	WaitPositionRequestTRIG := FALSE;
END_IF
(*****************************************************************************************************************************)
(*****************************************************************************************************************************)

(* Valutazione se la formatura attiva è di tipo misto oppure no, in questo caso, avendo una sola tipologia di formatura assegnamo l'indice di formatura fisso a 1 *)
FormaturaAttivaMista := TFValutaSeFormaturaMista(Forming);//,1);
FormatureMultipleAttive := TFValutaFormatureMultipleAttivate(Forming);
(* Bilanciamento 1=1 con pwa sulle WorkArea *)
//IF pwa < 1 OR pwa >= MAXAREA THEN
//	pwa := 1;
//ELSE
//	pwa := pwa + 1;
//END_IF
(*****************************************************************************************************************************)
(* Set variabili per gestione prelievo pacco dal ribaltino *)
(*****************************************************************************************************************************)
(* Set variabile che mi determina la possibilità di prelevare il pacco *)
HandlingOKPrelievoPacco := ((HandlingRun AND RibaltinoExitOk) OR (RichiestaStartRibaltino AND InWaitPosition));
TFTimerSet(ADR(TimerDepositoContinuoPallet),3000,HandlingRun);
RibaltinoOKPerDepositoContinuo := TFTimerDone(ADR(TimerDepositoContinuoPallet));
AbilitaComandiAnticipatiRibaltino := FROM_HMI_PAL.HMI_AbilitaComandiAnticipatiRibaltino;

(*****************************************************************************************************************************)
(*****************************************************************************************************************************)

(* Gestione e Creazione Missione per Ciclo Di Riposo*)
CASE WorkAreaManager^.State OF
	WAMANAGER_NOP:
			
		IF WaitPositionRequest AND 
		((NOT ForzaPrelievoPaccoDuranteCicloDiRiposo AND HandlingOKPrelievoPacco) OR 
		NOT ForzaPrelievoPaccoDuranteCicloDiRiposo OR 
		NOT HandlingOKPrelievoPacco OR 
		ExternalWaitPositionRequest OR 
		CicloDiRiposoNecessario) THEN
			WorkAreaManager^.State := WAMANAGER_CICLO_RIPOSO_INIT;
		END_IF
	
	WAMANAGER_CICLO_RIPOSO_INIT:
	
		Z_Riposo := QuotaFuoriIngombro_Z_AVUOTO; 			
	
		Mission^.PPick			:= PICKPOINT1;
		Mission^.TPick 			:= TPICK_NOT_DEFINED;
		Mission^.XPick			:= X_Riposo;
		Mission^.YPick			:= Y_Riposo;
		Mission^.ZPick			:= Z_Riposo;
		Mission^.JPick			:= J_Riposo;
		Mission^.JPickLT		:= PICKLTRESTPOSITION; // LONGITUDINALE
		Mission^.JPickVO		:= VORESTPOSITION;
		IF K_Riposo + PickPlaceParameters^.OffsetKPickPack < AxisPar_K.MinPosition THEN
			Mission^.KPick			:= AxisPar_K.MinPosition;
		ELSIF K_Riposo + PickPlaceParameters^.OffsetKPickPack > AxisPar_K.MaxPosition THEN
			Mission^.KPick			:= AxisPar_K.MaxPosition;
		ELSE
			Mission^.KPick			:= K_Riposo + PickPlaceParameters^.OffsetKPickPack;
		END_IF
		Mission^.KPickTorque	:= TORQUERESTPOSITION;
		Mission^.KPickMode 		:= KPICKMODERESTPOSITION;
		
		Mission^.PPlace			:= Mission^.PPick;
		Mission^.XPlace			:= Mission^.XPick;
		Mission^.YPlace			:= Mission^.YPick;
		Mission^.ZPlace			:= Mission^.ZPick;
		Mission^.JPlace			:= Mission^.JPick;	
		Mission^.KPlace			:= Mission^.KPick;
		
		WorkAreaManager^.State  := WAMANAGER_CICLO_RIPOSO_RUN;
		
	WAMANAGER_CICLO_RIPOSO_RUN:
	
		IF WorkPickPointState^[1].State=1  AND HandlingOKPrelievoPacco THEN
			PaccoSuRibaltinoDuranteCicloRiposo := TRUE;
			IF AbilitaForzaturaStatoDaRiposoAPrelievo^ AND NOT ExternalWaitPositionRequest AND NOT CicloDiRiposoNecessario AND FALSE THEN //Forzatura passaggio di stato
				ForzaPrelievoPaccoDuranteCicloDiRiposo := TRUE;
				WorkAreaManager^.State := WAMANAGER_SALTA_DA_RIPOSO_A_PRELIEVO;
			END_IF
		ELSE
			ForzaPrelievoPaccoDuranteCicloDiRiposo := FALSE;
			PaccoSuRibaltinoDuranteCicloRiposo := FALSE;
		END_IF
		
		IF Mission^.State = MISSION_STATE_VAIaRIPOSO_RUN THEN
			;
		ELSIF Mission^.State = MISSION_STATE_VAIaRIPOSO_END THEN
			CicloDiRiposoNecessario := FALSE;
			WorkAreaManager^.State 	:= WAMANAGER_CICLO_RIPOSO_END;	// setto lo stato del WAMANAGER
		ELSIF Mission^.State = MISSION_STATE_ERROR THEN
			;
		END_IF
		
	WAMANAGER_CICLO_RIPOSO_END:
		WorkAreaManager^.State := WAMANAGER_NOP;
		
	WAMANAGER_SALTA_DA_RIPOSO_A_PRELIEVO:
		IF Mission^.State = MISSION_STATE_VAIaRIPOSO_END THEN
			//ForzaPrelievoPaccoDuranteCicloDiRiposo := FALSE;
			WorkAreaManager^.State 	:= WAMANAGER_NOP;	// setto lo stato del WAMANAGER
		END_IF
						
END_CASE


IF WaitPositionRequest THEN
	FOR wapick := 1 TO MAXAREA DO
		IF AbilitaComandiAnticipatiRibaltino AND NOT FormaturaAttivaMista (*AND NOT FormatureMultipleAttive*) THEN
			(* Valutazione Presenza pacco su ribaltino e Comando in base a ........*)
			NumeroRibaltinoOccupatoConCodicePiazzola := TFPalletizerGetWPPFromPackCode(WorkPickPointState,WorkArea^[wapick].Code);
			ConsentiMovimentoRibaltino := (TFConsentiDepositoPaccoSuWA(WorkArea,WorkAreaState,wapick)AND FormaturaAttivaMista) OR NOT FormaturaAttivaMista;
			IF NumeroRibaltinoOccupatoConCodicePiazzola > 0 THEN
				IF WorkAreaManager^.State = WAMANAGER_CICLO_DEPOSITO_PACCO_RUN AND Mission^.PPlace = cwa AND 
					WorkArea^[Mission^.PPlace].Code = WorkPickPointState^[NumeroRibaltinoOccupatoConCodicePiazzola].Code AND FormaturaAttivaMista THEN
						IF Forming^[WorkAreaState^[Mission^.PPlace].F].PackXP[(WorkAreaState^[Mission^.PPlace].P)+ 1].Grip = -1 OR 
							Forming^[WorkAreaState^[Mission^.PPlace].F].PackXN[(WorkAreaState^[Mission^.PPlace].P)+ 1].Grip = -1 THEN
								ConsentiMovimentoRibaltino := FALSE; 
						END_IF
				END_IF
				IF ((NOT WaitPositionRequest AND FormaturaAttivaMista) OR NOT FormaturaAttivaMista) AND
					ConsentiMovimentoRibaltino AND HandlingRun THEN //AND WorkPickPointState^[NumeroRibaltinoOccupatoConCodicePiazzola].TS = 0 THEN
						IF NumeroRibaltinoOccupatoConCodicePiazzola > 0 AND Forming^[WorkAreaState^[wapick].F].Enable = 1 THEN // se c'è un pacco e i trasporti (quindi il ribaltino )sono in automatico
							(* Se il grip = -1 metto la Workarea nello stato WORKAREA_STATE_OCCUPIED_WORKED*)
							IF Forming^[WorkAreaState^[wapick].F].PackXP[WorkAreaState^[wapick].P].Grip = -1 OR
								Forming^[WorkAreaState^[wapick].F].PackXN[WorkAreaState^[wapick].P].Grip = -1 THEN
								//WorkPickPointState^[NumeroRibaltinoOccupatoConCodicePiazzola].TC := RIBALTINO_NOP;
							ELSE
								IF WorkPickPointState^[NumeroRibaltinoOccupatoConCodicePiazzola].TS = 0 AND WorkPickPointState^[NumeroRibaltinoOccupatoConCodicePiazzola].TC = 0  THEN
									IF WorkAreaState^[wapick].PN = 0 THEN							
										WorkPickPointState^[NumeroRibaltinoOccupatoConCodicePiazzola].TC := Forming^[WorkAreaState^[wapick].F].PackXP[WorkAreaState^[wapick].P].Grip + 1;	// Tipo di disposizione del pacco sul ribaltino
										UltimaPoastazioneDiAssegnazione := wapick;
										UltimoComando := Forming^[WorkAreaState^[wapick].F].PackXP[WorkAreaState^[wapick].P].Grip + 1;
										UltimoStatoCMDRibaltino := WorkAreaManager^.State;
										IF cmd >= 10 THEN
											cmd:=1;
										ELSE
											ComandoPickPoint[cmd] := WorkPickPointState^[1].TC;
											StatoPickPoint[cmd] := WorkPickPointState^[1].TS;
											cmd := cmd+1;
										END_IF
									ELSE
										WorkPickPointState^[NumeroRibaltinoOccupatoConCodicePiazzola].TC := Forming^[WorkAreaState^[wapick].F].PackXN[WorkAreaState^[wapick].P].Grip + 1;	// Tipo di disposizione del pacco sul ribaltino
										UltimaPoastazioneDiAssegnazione := wapick;
										UltimoComando := Forming^[WorkAreaState^[wapick].F].PackXN[WorkAreaState^[wapick].P].Grip + 1;
										UltimoStatoCMDRibaltino := WorkAreaManager^.State;
										IF cmd >= 10 THEN
											cmd:=1;
										ELSE
											ComandoPickPoint[cmd] := WorkPickPointState^[1].TC;
											StatoPickPoint[cmd] := WorkPickPointState^[1].TS;
											cmd := cmd+1;
										END_IF
									END_IF
								END_IF
							END_IF
						ELSE
							;
						END_IF
				END_IF
			END_IF
		END_IF
	END_FOR
END_IF



(*Con Stop in Fase, solo se la Missione è NOP vado in WAIT *)
IF NOT WaitPositionRequest OR 
	(WaitPositionRequest AND WorkAreaManager^.State <> WAMANAGER_NOP AND WorkAreaManager^.State <> WAMANAGER_CICLO_RIPOSO_RUN  AND WorkAreaManager^.State <> WAMANAGER_CICLO_RIPOSO_INIT) OR
	(WorkAreaManager^.State = WAMANAGER_NOP AND ForzaPrelievoPaccoDuranteCicloDiRiposo) THEN
	WAPointer := TFGetNearestWA(WorkArea,WorkPickPoint^[PICKPOINT1]);
	FOR pwa:=1 TO MAXAREA DO
		
		pwa := RestoringCWA(RestoreCWA,PreviousPWA,pwa);
		RestoreCWA^ := FALSE;		
		cwa := WAPointer[pwa].cwa;
		IF PreviousStackWA^ < 0 THEN
			PreviousStackWA^ := 1;
		END_IF
		IF cwa > 0 THEN
			;
		ELSE
			CONTINUE;
		END_IF
		
		IF AbilitaComandiAnticipatiRibaltino AND ((WorkAreaManager^.State <> WAMANAGER_CICLO_DEPOSITO_PACCO_RUN AND WorkAreaManager^.State <> WAMANAGER_CICLO_DEPOSITO_PACCO_END AND FormaturaAttivaMista) OR NOT FormaturaAttivaMista) THEN
			(* Valutazione Presenza pacco su ribaltino e Comando in base a ........*)
			NumeroRibaltinoOccupatoConCodicePiazzola := TFPalletizerGetWPPFromPackCode(WorkPickPointState,WorkArea^[cwa].Code);
			ConsentiMovimentoRibaltino := (TFConsentiDepositoPaccoSuWA(WorkArea,WorkAreaState,cwa)AND FormaturaAttivaMista) OR NOT FormaturaAttivaMista;
			IF NumeroRibaltinoOccupatoConCodicePiazzola > 0 THEN
				IF WorkAreaManager^.State = WAMANAGER_CICLO_DEPOSITO_PACCO_RUN AND Mission^.PPlace = cwa AND 
					WorkArea^[Mission^.PPlace].Code = WorkPickPointState^[NumeroRibaltinoOccupatoConCodicePiazzola].Code AND FormaturaAttivaMista THEN
						IF Forming^[WorkAreaState^[Mission^.PPlace].F].PackXP[(WorkAreaState^[Mission^.PPlace].P)+ 1].Grip = -1 OR 
							Forming^[WorkAreaState^[Mission^.PPlace].F].PackXN[(WorkAreaState^[Mission^.PPlace].P)+ 1].Grip = -1 THEN
								ConsentiMovimentoRibaltino := FALSE; 
						END_IF
				END_IF
				IF ((NOT WaitPositionRequest AND FormaturaAttivaMista) OR NOT FormaturaAttivaMista) AND
					ConsentiMovimentoRibaltino AND HandlingRun THEN //AND WorkPickPointState^[NumeroRibaltinoOccupatoConCodicePiazzola].TS = 0 THEN
						IF NumeroRibaltinoOccupatoConCodicePiazzola > 0 AND Forming^[WorkAreaState^[cwa].F].Enable = 1 THEN // se c'è un pacco e i trasporti (quindi il ribaltino )sono in automatico
							(* Se il grip = -1 metto la Workarea nello stato WORKAREA_STATE_OCCUPIED_WORKED*)
							IF Forming^[WorkAreaState^[cwa].F].PackXP[WorkAreaState^[cwa].P].Grip = -1 OR
								Forming^[WorkAreaState^[cwa].F].PackXN[WorkAreaState^[cwa].P].Grip = -1 THEN
								//WorkPickPointState^[NumeroRibaltinoOccupatoConCodicePiazzola].TC := RIBALTINO_NOP;
							ELSE
								IF WorkPickPointState^[NumeroRibaltinoOccupatoConCodicePiazzola].TS = 0 AND WorkPickPointState^[NumeroRibaltinoOccupatoConCodicePiazzola].TC = 0  THEN
									IF WorkAreaState^[cwa].PN = 0 THEN							
										WorkPickPointState^[NumeroRibaltinoOccupatoConCodicePiazzola].TC := Forming^[WorkAreaState^[cwa].F].PackXP[WorkAreaState^[cwa].P].Grip + 1;	// Tipo di disposizione del pacco sul ribaltino
										UltimaPoastazioneDiAssegnazione := cwa;
										UltimoComando := Forming^[WorkAreaState^[cwa].F].PackXP[WorkAreaState^[cwa].P].Grip + 1;
										UltimoStatoCMDRibaltino := WorkAreaManager^.State;
										IF cmd >= 10 THEN
											cmd:=1;
										ELSE
											ComandoPickPoint[cmd] := WorkPickPointState^[1].TC;
											StatoPickPoint[cmd] := WorkPickPointState^[1].TS;
											cmd := cmd+1;
										END_IF
									ELSE
										WorkPickPointState^[NumeroRibaltinoOccupatoConCodicePiazzola].TC := Forming^[WorkAreaState^[cwa].F].PackXN[WorkAreaState^[cwa].P].Grip + 1;	// Tipo di disposizione del pacco sul ribaltino
										UltimaPoastazioneDiAssegnazione := cwa;
										UltimoComando := Forming^[WorkAreaState^[cwa].F].PackXN[WorkAreaState^[cwa].P].Grip + 1;
										UltimoStatoCMDRibaltino := WorkAreaManager^.State;
										IF cmd >= 10 THEN
											cmd:=1;
										ELSE
											ComandoPickPoint[cmd] := WorkPickPointState^[1].TC;
											StatoPickPoint[cmd] := WorkPickPointState^[1].TS;
											cmd := cmd+1;
										END_IF
									END_IF
								END_IF
							END_IF
						ELSE
							;
						END_IF
				END_IF
			END_IF
		END_IF
		
		
		
		
		CASE WorkAreaState^[cwa].State OF
		
			(* Nota Piazzola VS PickPacco/PickPallet Vuoto da Catasta o PickFalda:
				1) E' la Piazzola Master che assegna la missione verso il ROBOT (* Missione Pick+Place *)
				2) La missione Termina dopo il Place
				3) Se si cancella la missione, la piazzola riprende d P
				4) Se c'è una missione e la piazzola diventa indisponibile si genera errore
			*)
			(* Se il Robot ha una missione "Pick/Place PALLET" destinata ad una piazzola che non è WORKAREA_STATE_FREE_WORKING si deve forzare un errore! *)
			(* Se il Robot ha una missione "Pick/Place PACCO" o "Pick/Place FALDA" destinata ad una piazzola che non è WORKAREA_STATE_OCCUPIED_WORKING si deve forzare un errore! *)
			
			(* Nota Puntatore Formatura: -1=Inizio Lavorazione, 0=Gestione Eventuale Falda Dopo Pallet, 1..n=Gestione Pacchi/Falde dopo Strato *)
			(* ******************************************************************************************************** *)
			(* ******************************************************************************************************** *)
				(* Free + Disabled *)
			WORKAREA_STATE_FREE_DISABLED:
				(* Valuto il numero dei pacchi sulla linea e se è possibile depositare i pallet di continuo *)
				NPacchiPresentiSuLinea := TFNumeroPacchiSuLinea(ArrayPacchi);
				NUltimiTrasportiOccupati := TFNumeroUltimi_N_TrasportiOccupati(ArrayPacchi,12);//FROM_HMI_PAL.HMI_NumeroPacchiMassimoDepositoPalletContinuo);
				OKDepositoPalletContinuo := AbilitaDisposizionePalletContinua^ AND RibaltinoOKPerDepositoContinuo AND NOT FormatureMultipleAttive AND 
											TFDepositoContinuoPalletConsentito(NpacchiPresenti:=NPacchiPresentiSuLinea,NpacchiMassimiConsentiti:=FROM_HMI_PAL.HMI_NumeroPacchiMassimoDepositoPalletContinuo,NultimiTrasportiOccupati:=NUltimiTrasportiOccupati);
				(* Cerco se ci sono già dei pallet depositati in attesa di ricevere il codice *)
				PalletDepositatiSenzaCodicePresenti := TFPalletizerIsCodeAssigned(WorkArea,WorkAreaState,0);
				(* Si verifica se Jolly o no e si passa in WORKING. Se Jolly si cerca codice non assegnato *)
				IF WorkArea^[cwa].Enable = 1 THEN
					IF WorkAreaState^[cwa].P = -1  THEN
						(* Per Pallet si attiva solo se il codice assegnato è un dato valido *)
						IF WorkArea^[cwa].Typology = TYPOLOGY_PALLET THEN
							(* Postazione Zona *)
							IF TFPalletizerIsWorkAreaIntoZone(WorkAreaZone,cwa) AND GestioneAZoneAbilitata^ THEN                     // Se la WA appartiene a una zona
								pcode := TFPackCodePresenteInZona(WorkPickPointState:=WorkPickPointState,WorkAreaZone:=WorkAreaZone,WorkArea:=cwa);//Il codice del pacco sul ribaltino appartiene alla zona della postazione in esame
								(* Cerco Formatura *)
								fcode := TFPalletizerGetFormingFromCode(Forming,pcode);
								IF NOT FormatureMultipleAttive THEN //Se NON ci sono più formature Diverse Abilitate valuto i codici non assegnati e li dispongo
									pcodeUnassigned := TFPalletizerGetUnassignedCode(WorkArea,WorkAreaState,Forming);
									(* Cerco Formatura *)
									IF pcodeUnassigned > 0 THEN
										fcode := TFPalletizerGetFormingFromCode(Forming,pcodeUnassigned);
									END_IF
								ELSE
									pcodeUnassigned :=0;
								END_IF
								
								IF (pcode > 0 OR pcodeUnassigned > 0)THEN 
									(* Se ho trovato un codice non assegnato e ho l'abilitazione del deposito continuo attivo e l'ok per il deposito *)
									IF pcodeUnassigned > 0 AND OKDepositoPalletContinuo THEN
										fcode := TFPalletizerGetFormingFromCode(Forming,pcodeUnassigned);
										IF fcode > 0 THEN
											CicloDiRiposoNecessario := FALSE;	
											WorkArea^[cwa].Taped := -1;
											WorkArea^[cwa].LGV_ReqAbort := FALSE;
											IF AbilitaAssegnazioneCodicePiazzoleConPaccoSuRibaltino THEN
												WorkArea^[cwa].Code := 0;
												WorkArea^[cwa].Initialize := TRUE;
											ELSE
												WorkArea^[cwa].Code := pcodeUnassigned;
												WorkArea^[cwa].Initialize := FALSE;
												pcodeUnassigned := 0;
											END_IF
											WorkAreaState^[cwa].F := fcode;
											WorkAreaState^[cwa].P := -1;
											WorkAreaState^[cwa].L := -1;
											WorkAreaState^[cwa].PN := -1;
											WorkAreaState^[cwa].LGVAttr := Forming^[WorkAreaState^[cwa].F].LGVAttr;
											WorkAreaState^[cwa].State := WORKAREA_STATE_FREE_WORKING;
										ELSE
											// Errore
										END_IF
									(* Se NON ho nessuna piazzola in lavorazione con il codice di lavorazione e il codice di formatura già PRESENTI e IN LAVORAZIONE
									 o posso depositare il pallet in continuazione *)
									ELSIF ((*NOT TFPalletizerIsCodeAssigned(WorkArea,WorkAreaState,pcode) AND*) NOT TFPalletizerIsFormingAssigned(FCode:=fcode,WorkArea:=WorkArea,WorkAreaState:=WorkAreaState,PCode:=pcode)) THEN
										(* Cerco Formatura *)
										fcode := TFPalletizerGetFormingFromCode(Forming,pcode);
										IF fcode > 0 AND pcode > 0 THEN
											CicloDiRiposoNecessario := FALSE;
											WorkArea^[cwa].Taped := -1;
											WorkArea^[cwa].LGV_ReqAbort := FALSE;
											IF AbilitaAssegnazioneCodicePiazzoleConPaccoSuRibaltino THEN
												WorkArea^[cwa].Code := 0;
												WorkArea^[cwa].Initialize := TRUE;
											ELSE
												WorkArea^[cwa].Code := pcode;
												WorkArea^[cwa].Initialize := FALSE;
												pcode := 0;
											END_IF
											WorkAreaState^[cwa].F := fcode;
											WorkAreaState^[cwa].P := -1;
											WorkAreaState^[cwa].L := -1;
											WorkAreaState^[cwa].PN := -1;
											WorkAreaState^[cwa].LGVAttr := Forming^[WorkAreaState^[cwa].F].LGVAttr;
											WorkAreaState^[cwa].State := WORKAREA_STATE_FREE_WORKING;
										ELSE
											;// Errore
										END_IF
									END_IF
								END_IF
							ELSE
								;(* Postazione Assegnata Con codice Fisso *)								
								(*IF WorkArea^[cwa].Jolly <> 1 AND OKDepositoPalletContinuo THEN
									IF WorkArea^[cwa].Code > 0 (*AND OKDepositoPalletContinuo*) THEN
										(* Cerco Formatura *)
										fcode := TFPalletizerGetFormingFromCode(Forming,WorkArea^[cwa].Code);
										IF fcode > 0 THEN
											CicloDiRiposoNecessario := FALSE;	
											WorkArea^[cwa].Taped := -1;
											WorkArea^[cwa].LGV_ReqAbort := FALSE;
											WorkAreaState^[cwa].F := fcode;
											WorkAreaState^[cwa].P := -1;
											WorkAreaState^[cwa].L := -1;
											WorkAreaState^[cwa].PN := -1;
											WorkAreaState^[cwa].LGVAttr := Forming^[WorkAreaState^[cwa].F].LGVAttr;
											WorkAreaState^[cwa].State := WORKAREA_STATE_FREE_WORKING;
										ELSE
											// Errore
										END_IF
									END_IF
								ELSE
									(* Postazione Jolly: Il codice viene assegnato valutando i codici sulla linea *)
									(* Se Jolly si Attiva se si trova un codice da assegnare *)
									// pcode := TFPalletizerGetUnassignedCode(WorkArea,WorkAreaState,Forming);
									pcode := TFPackCodePresenteInWAJolly(ArrayPacchi:=ArrayPacchi,WorkArea:=WorkArea,WorkAreaState:=WorkAreaState);//TFPackCodePresentToJollyWorkArea(HandlingPackTable,WorkArea,WorkAreaState);
									IF pcode > 0 THEN
										fcode := TFPalletizerGetFormingFromCode(Forming,pcode);
										IF fcode > 0 THEN
											WorkArea^[cwa].Taped := -1;
											WorkArea^[cwa].LGV_ReqAbort := FALSE;
											IF AbilitaAssegnazioneCodicePiazzoleConPaccoSuRibaltino THEN
												WorkArea^[cwa].Code := 0;
												WorkArea^[cwa].Initialize := TRUE;
											ELSE
												WorkArea^[cwa].Code := pcode;
												WorkArea^[cwa].Initialize := FALSE;
												pcode := 0;
											END_IF
											WorkAreaState^[cwa].F := fcode;
											WorkAreaState^[cwa].P := -1;
											WorkAreaState^[cwa].L := -1;
											WorkAreaState^[cwa].PN := -1;
											WorkAreaState^[cwa].LGVAttr := Forming^[WorkAreaState^[cwa].F].LGVAttr;
											WorkAreaState^[cwa].State := WORKAREA_STATE_FREE_WORKING;
										ELSE
											// Errore
										END_IF
									ELSE
										;
									END_IF
								END_IF*)
							END_IF
						ELSE (* Per Cataste o Falde si Attiva senza controlli *)
							WorkArea^[cwa].Taped := -1;
							//WorkArea^[cwa].Learned_Z := WorkArea^[cwa].Learn_Z;
							//WorkArea^[cwa].H := 1000;
							WorkAreaState^[cwa].P := -1;
							WorkAreaState^[cwa].L := -1;
							WorkAreaState^[cwa].PN := -1;
							IF PX_WorkArea[cwa] THEN // Con presenza vado in lavorazione altrimenti forzo chiamata LGV
								WorkAreaState^[cwa].State := WORKAREA_STATE_OCCUPIED_WORKING;
							ELSE
								WorkAreaState^[cwa].State := WORKAREA_STATE_OCCUPIED_ENDED;
							END_IF							
						END_IF
					ELSE
						WorkAreaState^[cwa].State := WORKAREA_STATE_OCCUPIED_WORKING;
					END_IF;	
			ELSE
				;
			END_IF
(**********************************************************************************************************************************************************************************)
(**********************************************************************************************************************************************************************************)
			(* Occupied + Disabled *)
(**********************************************************************************************************************************************************************************)
(**********************************************************************************************************************************************************************************)
			WORKAREA_STATE_OCCUPIED_DISABLED:
				(* Nessuna Operazione! Si PROSEGUE LA LAVORAZIONE se viene Abilitata la Piazzola *)
				IF WorkArea^[cwa].Enable = 1  AND  Forming^[WorkAreaState^[cwa].F].Enable = 1 THEN
					WorkAreaState^[cwa].State := WORKAREA_STATE_OCCUPIED_WORKING;
				END_IF
	
			(* Free + Working (Gestione PALLET VUOTO) *)
			WORKAREA_STATE_FREE_WORKING:
				IF PreviousStackWA^ < 0 THEN
					PreviousStackWA^ := 1;
				END_IF
				IF WorkArea^[cwa].Enable = 1 THEN //oR (WorkArea^[cwa].Enable = 0 AND Mission^.State > MISSION_STATE_NOP) THEN
					(* 	1) Se Nessuna Missione in Corso (Mission.State=NOP) allora eseguo i punti sotto
						2) Verifica Catasta Disponibile per Prelievo Pallet. Se SI Proseguo altrimenti nulla
						3) Creo Missione Pick/Place Pallet e assegno Mission.State = MISSION_STATE_PICKING
						4) Con Mission.State = MISSION_STATE_PICKED o MISSION_STATE_PLACING non si fa nulla
						5) Con Mission.State = MISSION_STATE_PLACED e PlaceID della Missione è QUESTA WorkArea la Missione Passa a NOP per liberare il Gestore
						6) Assegno WorkArea^[cwa].P=0 per inizio Pallettizzazione + WorkArea^[cwa].L=0 per deposito prima Falda *)
					CASE WorkAreaManager^.State OF
						WAMANAGER_NOP:
						
							(* Cerco disponibilità Pallet *)
							IF TFPalletizerIsStackAvailable(WorkArea,WorkAreaState,PreviousStackWA,Forming^[WorkAreaState^[cwa].F].Pallet) THEN
								ppick := PreviousStackWA^;
							ELSE	
								ppick := TFPalletizerGetWAFromTypeCode(WorkArea,WorkAreaState,TYPOLOGY_STACK,Forming^[WorkAreaState^[cwa].F].Pallet);
								PreviousStackWA^ := ppick; 
							END_IF
							
							IF ppick <> -1 THEN
								CicloDiRiposoNecessario := FALSE;
								IF ppick > 0 AND 										// esiste una catasta pallatte con codice idoneo alle formature attive 
									PX_WorkArea[ppick] AND 								// la fotocellula di presenza catasta è indica l'effettiva presenza dei pallet
									WorkArea^[cwa].Typology <> TYPOLOGY_STACK THEN 		// la tipologia della workarea che devo valurtare NON è di tipo catasta vuoti
									IF 	Forming^[WorkAreaState^[cwa].F].Layer > 0 AND 	// La formatura richiede la falda sopra il pallet
										WorkAreaState^[cwa].L <= 0 THEN 				// il pallet sulla catasta non ha già la falda depositata	
										(* Cerco se è presente una piazzola adibita a magazzino falde con codice presente in formtura*)
										lpick := TFPalletizerGetWAFromTypeCode(WorkArea,WorkAreaState,TYPOLOGY_LAYER,Forming^[WorkAreaState^[cwa].F].Layer); // mi restituisce il numero della piazzola adibita a magazzino falda del codice richiesto
										IF lpick <> -1 THEN
											IF lpick > 0 AND 			// se c'è un magazzino falde con codice ok
												PX_WorkArea[lpick]THEN	// se la fotocellula del magazzino mi indica l'effettiva presenza delle falde (=> magazzino NON vuoto!)
												WorkAreaManager^.State  := WAMANAGER_CICLO_FALDA_VUOTI_INIT;	// setto lo stato del WAMANAGER
												RestoreCWA^ := TRUE;
												PreviousPWA^ := pwa;
												EXIT;
											END_IF
										END_IF	
									ELSE
										WorkAreaManager^.State 	:= WAMANAGER_CICLO_PALL_INIT;
										RestoreCWA^ := TRUE;
										PreviousPWA^ := pwa;
										EXIT;
									END_IF
								END_IF
							ELSE
							//;	CicloDiRiposoNecessario := TRUE;
							END_IF
							(* Creo Missione Falda per deposito su catasta vuoti *)
						WAMANAGER_CICLO_FALDA_VUOTI_INIT:
						
							Mission^.PPick			:= lpick;
							Mission^.TPick 			:= TPICK_LAYER;
							Mission^.PPlace			:= ppick;
							Mission^.XPick			:= WorkArea^[Mission^.PPick].X + WorkAreaOffset^[Mission^.PPick].X;//+ (Layer^[WorkArea^[Mission^.PPick].Layer].X / 2);
							CASE TIPO_MAGAZZINO_FALDE OF
								MAGAZZINO_FALDE_CENTRO_FISSO:
									Mission^.YPick			:= WorkArea^[Mission^.PPick].Y + WorkAreaOffset^[Mission^.PPick].Y;// + (Layer^[WorkArea^[Mission^.PPick].Layer].Y / 2);
								MAGAZZINO_FALDE_CENTRO_VARIABILE:
									Mission^.YPick			:= WorkArea^[Mission^.PPick].Y + WorkAreaOffset^[Mission^.PPick].Y + (Layer^[WorkArea^[Mission^.PPick].Layer].Y / 2);
							END_CASE
							
							//IF  WorkArea^[Mission^.PPick].DoLearn_Z = 1 THEN				// se DEVO efettuare l'apprendimento
								//Mission^.ZPick	:= WorkArea^[Mission^.PPick].Learn_Z; 	// Quota di inizio apprendimento
							//ELSE														// se NON DEVO efettuare l'apprendimento (cilo successivo al primo!! o dopo Richiesta Ingresso)
								Mission^.ZPick	:= WorkArea^[Mission^.PPick].Z + WorkAreaOffset^[Mission^.PPick].Z; (*+ WorkArea^[Mission^.PPick].H;*) (* Posizione WorkArea + Altezza Reale *) // in questo modo LA LENTA va sempre fino a zero...mi fermo al raggiungimento dell'intervento dei tastatori
							//END_IF
							Mission^.JPick			:= WorkArea^[Mission^.PPick].JPick + WorkAreaOffset^[Mission^.PPick].J;
							Mission^.KPick			:= Pallet^[WorkArea^[Mission^.PPlace].Pallet].X; (* + PickPlaceParameters^.OffsetKPick; *)
							Mission^.KPickTorque	:= KPICKTORQUELAYER;
							Mission^.KPickMode 		:= KSUCTIONMODE;
							Mission^.XPlace			:= WorkArea^[Mission^.PPlace].X + WorkAreaOffset^[Mission^.PPlace].X;
							Mission^.YPlace			:= WorkArea^[Mission^.PPlace].Y + WorkAreaOffset^[Mission^.PPlace].Y + (Pallet^[Forming^[WorkAreaState^[cwa].F].Pallet].Y / 2);
							IF  WorkArea^[Mission^.PPlace].DoLearn_Z = 1 THEN 	// se devo fare l'apprendimento sulla catasta vuoti
								//Mission^.ZPlace		:= WorkArea^[Mission^.PPlace].Learn_Z; //quota inizio apprendimento catasta vuoti
								Mission^.ZPlace	:= WorkArea^[Mission^.PPlace].Z + WorkAreaOffset^[Mission^.PPlace].Z; // in questo modo LA LENTA va sempre fino a zero...mi fermo al raggiungimento dell'intervento dei tastatori
							ELSE											// se NON devo fare l'apprendimento sulla catasta vuoti
								Mission^.ZPlace		:= WorkArea^[Mission^.PPlace].Z + WorkAreaOffset^[Mission^.PPlace].Z;// + WorkArea^[Mission^.PPlace].H; //quota reale catasta vuoti = (altezza WA + altezza reale)
							END_IF
							Mission^.JPlace			:= WorkArea^[Mission^.PPlace].JPlace + WorkAreaOffset^[Mission^.PPlace].J;
							Mission^.KPlace			:= Mission^.KPick;//WorkArea^[Mission^.PPick].KPick;//Layer^[WorkArea^[cwa].Layer].X + 20;
							Mission^.KPlaceMode 	:= KSUCTIONMODE;
							Mission^.XPlaceApproach	:= Mission^.XPlace + WorkAreaOffset^[Mission^.PPlace].X;
							Mission^.YPlaceApproach	:= Mission^.YPlace + WorkAreaOffset^[Mission^.PPlace].Y;
							Mission^.ZPlaceApproach	:= Mission^.ZPlace + WorkAreaOffset^[Mission^.PPlace].Z;
							Mission^.JPlaceApproach	:= Mission^.JPlace + WorkAreaOffset^[Mission^.PPlace].J;
							Mission^.XDim			:= Layer^[Forming^[WorkAreaState^[cwa].F].Layer].X;
							Mission^.YDim			:= Layer^[Forming^[WorkAreaState^[cwa].F].Layer].Y;
							Mission^.ZDim			:= Layer^[Forming^[WorkAreaState^[cwa].F].Layer].Z;
							WorkAreaManager^.State 	:= WAMANAGER_CICLO_PRELIEVO_FALDA_VUOTI_RUN;
							EXIT;
												
						WAMANAGER_CICLO_PRELIEVO_FALDA_VUOTI_RUN:
	
							IF Mission^.State = MISSION_STATE_PRELIEVO_FALDA_RUN THEN
								;
							ELSIF Mission^.State = MISSION_STATE_PRELIEVO_FALDA_END THEN
								WorkAreaManager^.State 	:= WAMANAGER_CICLO_PRELIEVO_FALDA_VUOTI_END;	// setto lo stato del WAMANAGER
								EXIT;
							ELSIF Mission^.State = MISSION_STATE_ERROR THEN
								;
							END_IF
							
						WAMANAGER_CICLO_PRELIEVO_FALDA_VUOTI_END:	
							IF Mission^.TPick = TPICK_LAYER THEN
								IF WorkArea^[Mission^.PPick].Typology = TYPOLOGY_LAYER THEN
									IF WorkArea^[Mission^.PPick].H > (WorkArea^[Mission^.PPick].Z + WorkAreaOffset^[Mission^.PPick].Z + Layer^[WorkArea^[Mission^.PPick].Layer].Z) THEN
										WorkArea^[Mission^.PPick].H := ModuleAX_Z^.Ax^.Status.ActPosition; (*- WorkArea^[Mission^.PPick].Z;*)//WorkArea^[Mission^.PPick].H - Layer^[WorkArea^[Mission^.PPick].Layer].Z;
										WorkArea^[Mission^.PPick].DoLearn_Z := 2;
										WorkArea^[Mission^.PPick].Learned_Z := ModuleAX_Z^.Ax^.Status.ActPosition;
									ELSE
										WorkArea^[Mission^.PPick].H := 0;
										WorkArea^[Mission^.PPick].DoLearn_Z := 1;
										//WorkAreaState^[Mission^.PPick].State := WORKAREA_STATE_OCCUPIED_ENDED;	
									END_IF
								
								END_IF
							END_IF
							WorkAreaManager^.State 	:= WAMANAGER_CICLO_DEPOSITO_FALDA_VUOTI_RUN;	// setto lo stato del WAMANAGER
							EXIT;
	
						WAMANAGER_CICLO_DEPOSITO_FALDA_VUOTI_RUN:	
							IF Mission^.State = MISSION_STATE_DEPOSITO_FALDA_RUN THEN
								;
							ELSIF Mission^.State = MISSION_STATE_DEPOSITO_FALDA_END THEN
								WorkAreaManager^.State 	:= WAMANAGER_CICLO_DEPOSITO_FALDA_VUOTI_END;	// setto lo stato del WAMANAGER
								EXIT;
							ELSIF Mission^.State = MISSION_STATE_ERROR THEN
								;
							END_IF
							
						WAMANAGER_CICLO_DEPOSITO_FALDA_VUOTI_END:
							WorkAreaState^[Mission^.PPlace].L := 1;								// setto la presenza della falda sul pallet
							
							IF WorkArea^[Mission^.PPlace].DoLearn_Z = 1 THEN			// se sulla piazzola era da effettuare l'apprendimento
								WorkArea^[Mission^.PPlace].Learned_Z := ModuleAX_Z^.Ax^.Status.ActPosition - (WorkArea^[Mission^.PPlace].Z + WorkAreaOffset^[Mission^.PPlace].Z);				// set della quota rilevata durante apprndimento
								WorkArea^[Mission^.PPlace].DoLearn_Z := 2;				// setto l' vvenuto apprendimento della quota della catasta pallet 
								WorkArea^[Mission^.PPlace].H := WorkArea^[Mission^.PPlace].Learned_Z;
							END_IF
							
							RestoreCWA^ := TRUE;
							PreviousPWA^ :=cwa;
							WorkAreaManager^.State 	:= WAMANAGER_CICLO_PALL_INIT;
							EXIT;
							
						(* Creo Missione Pallet per deposito su piazzola*)
						WAMANAGER_CICLO_PALL_INIT:
							Mission^.PPick			:= ppick;
							Mission^.TPick 			:= TPICK_PALLET;
							Mission^.PPlace			:= cwa;
							Mission^.XPick			:= WorkArea^[Mission^.PPick].X + WorkAreaOffset^[Mission^.PPick].X;
							Mission^.YPick			:= WorkArea^[Mission^.PPick].Y + WorkAreaOffset^[Mission^.PPick].Y + (Pallet^[WorkArea^[Mission^.PPick].Pallet].Y / 2);
							IF  WorkArea^[Mission^.PPick].DoLearn_Z = 1 THEN
								Mission^.ZPick	:= WorkArea^[Mission^.PPick].Z + WorkAreaOffset^[Mission^.PPick].Z;//WorkArea^[Mission^.PPlace].Z; // in questo modo LA LENTA va sempre fino a zero...mi fermo al raggiungimento dell'intervento dei tastatori
								//Mission^.ZPick	:= WorkArea^[Mission^.PPick].Learn_Z; (* Quota di START apprendimento *)
							ELSE
								Mission^.ZPick	:= WorkArea^[Mission^.PPick].Z + WorkAreaOffset^[Mission^.PPick].Z;// + WorkArea^[Mission^.PPick].H;//WorkArea^[Mission^.PPlace].Z + WorkArea^[Mission^.PPlace].H;//WorkArea^[Mission^.PPick].Z + WorkArea^[Mission^.PPick].H; (* Posizione WorkArea + Altezza Reale *)
							END_IF
							Mission^.JPick			:= WorkArea^[Mission^.PPick].JPick + WorkAreaOffset^[Mission^.PPick].J;
							Mission^.KPick			:= Pallet^[WorkArea^[Mission^.PPick].Pallet].X;
							Mission^.KPickTorque	:= PickPlaceParameters^.KPickTorquePallet;
							IF NOT SimulazioneSenzaPallet THEN //Se non sono in simulazione utilizzo la presa con coppia
								Mission^.KPickMode 		:= KTORQUEMODE;
							ELSE
								Mission^.KPickMode 		:= KPOSITIONMODE;
							END_IF
							Mission^.XPlace			:= WorkArea^[Mission^.PPlace].X + WorkAreaOffset^[Mission^.PPlace].X;
							Mission^.YPlace			:= WorkArea^[Mission^.PPlace].Y + WorkAreaOffset^[Mission^.PPlace].Y + (Pallet^[Forming^[WorkAreaState^[cwa].F].Pallet].Y / 2);
							Mission^.ZPlace			:= WorkArea^[Mission^.PPlace].Z + WorkAreaOffset^[Mission^.PPlace].Z + WorkArea^[Mission^.PPlace].H + Pallet^[Forming^[WorkAreaState^[cwa].F].Pallet].Z + PickPlaceParameters^.OffsetZPlacePallet;
							Mission^.JPlace			:= WorkArea^[Mission^.PPlace].JPlace + WorkAreaOffset^[Mission^.PPlace].J;
							Mission^.KPlace			:= Pallet^[Forming^[WorkAreaState^[cwa].F].Pallet].X; (*+ PickPlaceParameters^.OffsetKPlace;*)
							Mission^.KPlaceMode 	:= KPOSITIONMODE;
							Mission^.XPlaceApproach	:= Mission^.XPlace;
							Mission^.YPlaceApproach	:= Mission^.YPlace;
							Mission^.ZPlaceApproach	:= Mission^.ZPlace;
							Mission^.JPlaceApproach	:= Mission^.JPlace;
							Mission^.XDim			:= Pallet^[Forming^[WorkAreaState^[cwa].F].Pallet].X;
							Mission^.YDim			:= Pallet^[Forming^[WorkAreaState^[cwa].F].Pallet].Y;
							Mission^.ZDim			:= Pallet^[Forming^[WorkAreaState^[cwa].F].Pallet].Z;
							
							(* Valorizzo la variabile che serve per calolare la quota di fuori ingombro verticale della pinza *)
							IF AbilitaOffsetInUscitaTasteggioPrelievoPallet^ THEN // Se ho l'abilitazione dell'uscita dai tastatori con Offset
								Dimensione_Z_ElementoInPresaX_Ingombro := Mission^.ZDim + PickPlaceParameters^.OffsetZUscitaTasteggioPickPallet; // Se ho abilitato l'uscita con Offset dai tastatori lo aggiungo alla dimensione dell'elemento
							ELSE
								Dimensione_Z_ElementoInPresaX_Ingombro := Mission^.ZDim;
							END_IF
							
							RestoreCWA^ := TRUE;
							PreviousPWA^ := pwa;
								
							WorkAreaManager^.State 	:= WAMANAGER_CICLO_PRELIEVO_PALL_RUN;
							EXIT;
							
						WAMANAGER_CICLO_PRELIEVO_PALL_RUN:
							IF 	Mission^.State = MISSION_STATE_PRELIEVO_PALLET_RUN THEN
								;
							ELSIF Mission^.State = MISSION_STATE_PRELIEVO_PALLET_END THEN
								WorkAreaManager^.State 	:= WAMANAGER_CICLO_PRELIEVO_PALL_END;
								RestoreCWA^ := TRUE;
								PreviousPWA^ :=cwa;
								EXIT;
							ELSIF Mission^.State = MISSION_STATE_ERROR THEN
								;
							END_IF
							
						WAMANAGER_CICLO_PRELIEVO_PALL_END:	
								IF WorkArea^[Mission^.PPick].DoLearn_Z = 1 THEN 									// se stavo facendo l'apprendimento della quota
									WorkArea^[Mission^.PPick].Learned_Z := ModuleAX_Z^.Ax^.Status.ActPosition;	// set della quota rilevata durante apprndimento
									WorkArea^[Mission^.PPick].H := ModuleAX_Z^.Ax^.Status.ActPosition;//WorkArea^[Mission^.PPick].Learned_Z;
									WorkArea^[Mission^.PPick].DoLearn_Z := 2;
								END_IF
								IF (*WorkArea^[Mission^.PPick].H > Pallet^[WorkArea^[Mission^.PPick].Pallet].Z AND*) WorkArea^[Mission^.PPick].DoLearn_Z=2 THEN
									WorkArea^[Mission^.PPick].Learned_Z := ModuleAX_Z^.Ax^.Status.ActPosition;
								//WorkArea^[Mission^.PPick].H := WorkArea^[Mission^.PPick].H - Pallet^[WorkArea^[Mission^.PPick].Pallet].Z;
									WorkArea^[Mission^.PPick].H := ModuleAX_Z^.Ax^.Status.ActPosition;// WorkArea^[Mission^.PPick].Learned_Z;
									WorkArea^[Mission^.PPick].DoLearn_Z := 2;
								ELSE
									WorkArea^[Mission^.PPick].H := 0;				// a questo punto non ho più pallet, quindi altezza 0!!
									WorkArea^[Mission^.PPick].DoLearn_Z := 1;			// devo quindi effettuare l'apprendimento quando avrò la nuova catasta!!!
									WorkArea^[Mission^.PPick].Learned_Z := ALTEZZA_CATASTA_VUOTI;
								END_IF
								WorkAreaState^[Mission^.PPick].State := WORKAREA_STATE_OCCUPIED_ENDED;	
								WorkAreaManager^.State 	:= WAMANAGER_CICLO_DEPOSITO_PALL_RUN;
								EXIT;
								
						WAMANAGER_CICLO_DEPOSITO_PALL_RUN:	
							IF Mission^.State = MISSION_STATE_DEPOSITO_PALLET_RUN THEN
								;	
							ELSIF Mission^.State = MISSION_STATE_DEPOSITO_PALLET_END THEN
								WorkAreaManager^.State 	:= WAMANAGER_CICLO_DEPOSITO_PALL_END;
								RestoreCWA^ := TRUE;
								PreviousPWA^ :=cwa;
								EXIT;
							ELSIF Mission^.State = MISSION_STATE_ERROR THEN
								;
							END_IF
							
						WAMANAGER_CICLO_DEPOSITO_PALL_END:	
							/////////////////////////////
							(* X simulazione *)
							PalletPrelevatiXSimulazione := PalletPrelevatiXSimulazione+1;
							IF PalletPrelevatiXSimulazione >= PalletPrelevatiSimulazioneMAX THEN
								PalletPrelevatiXSimulazione := 0;
								I_PHPresenzaPalletVirtuale[Mission^.PPick] := FALSE;
							END_IF
							
							//////////////////////////////////////
							IF WorkAreaState^[Mission^.PPick].L < 0 THEN
								IF NOT HMI_AbilitaTasteggioDepositoPallet THEN // Se non ho abilitata la funzione di tasteggio in deposito pallet, setto le altezze con le altezze ideali
									WorkArea^[Mission^.PPlace].H := Pallet^[Forming^[WorkAreaState^[Mission^.PPlace].F].Pallet].Z;
									WorkArea^[Mission^.PPlace].HPL := Pallet^[Forming^[WorkAreaState^[Mission^.PPlace].F].Pallet].Z;
								ELSE	// Setto le altezze con la posizione attuale, cercando di aumentare la precisione in fase di deposito pacco
									WorkArea^[Mission^.PPlace].H := ModuleAX_Z^.Ax^.Status.ActPosition;
									WorkArea^[Mission^.PPlace].HPL := ModuleAX_Z^.Ax^.Status.ActPosition;
								END_IF
								WorkArea^[Mission^.PPlace].ProgressiveNr := ProgressiveNrWA^;
								ProgressiveNrWA^ := ProgressiveNrWA^ + 1;
								WorkAreaState^[Mission^.PPlace].P := 0;
								WorkAreaState^[Mission^.PPlace].L := 0;
								WorkArea^[Mission^.PPlace].Slow := 0;
								WorkAreaState^[Mission^.PPlace].LGVAttr := Forming^[WorkAreaState^[Mission^.PPlace].F].LGVAttr;
								WorkAreaState^[Mission^.PPlace].State := WORKAREA_STATE_OCCUPIED_WORKING;
								WorkAreaManager^.State 	:= WAMANAGER_NOP;
								RestoreCWA^ := TRUE;
								PreviousPWA^ :=cwa;
								I_PHPresenzaPalletVirtuale[Mission^.PPlace] := TRUE;
								EXIT;
							ELSE
								IF NOT HMI_AbilitaTasteggioDepositoPallet THEN // Se non ho abilitata la funzione di tasteggio in deposito pallet, setto le altezze con le altezze ideali
									WorkArea^[Mission^.PPlace].H := Pallet^[Forming^[WorkAreaState^[Mission^.PPlace].F].Pallet].Z + Layer^[Forming^[WorkAreaState^[Mission^.PPlace].F].Layer].Z;
									WorkArea^[Mission^.PPlace].HPL := Pallet^[Forming^[WorkAreaState^[Mission^.PPlace].F].Pallet].Z + Layer^[Forming^[WorkAreaState^[Mission^.PPlace].F].Layer].Z;
								ELSE	// Setto le altezze con la posizione attuale, cercando di aumentare la precisione in fase di deposito pacco
									IF AbilitaOffsetInUscitaTasteggioPrelievoPallet^ THEN // Se ho l'abilitazione dell'uscita dai tastatori con Offset
										WorkArea^[Mission^.PPlace].H := ModuleAX_Z^.Ax^.Status.ActPosition - PickPlaceParameters^.OffsetZUscitaTasteggioPickPallet;
										WorkArea^[Mission^.PPlace].HPL := ModuleAX_Z^.Ax^.Status.ActPosition - PickPlaceParameters^.OffsetZUscitaTasteggioPickPallet;
									ELSE
										WorkArea^[Mission^.PPlace].H := ModuleAX_Z^.Ax^.Status.ActPosition;
										WorkArea^[Mission^.PPlace].HPL := ModuleAX_Z^.Ax^.Status.ActPosition;
									END_IF
								END_IF
								WorkArea^[Mission^.PPlace].ProgressiveNr := ProgressiveNrWA^;
								ProgressiveNrWA^ := ProgressiveNrWA^ + 1;
								WorkAreaState^[Mission^.PPlace].P := 1;
								WorkAreaState^[Mission^.PPlace].L := 1;
								WorkArea^[Mission^.PPlace].Slow := 0;
								WorkAreaState^[Mission^.PPlace].LGVAttr := Forming^[WorkAreaState^[Mission^.PPlace].F].LGVAttr;
								WorkAreaState^[Mission^.PPlace].State := WORKAREA_STATE_OCCUPIED_WORKING;
								WorkAreaManager^.State 	:= WAMANAGER_NOP;
								RestoreCWA^ := TRUE;
								PreviousPWA^ :=cwa;
								I_PHPresenzaPalletVirtuale[Mission^.PPlace] := TRUE;
								EXIT;
							END_IF
							IF NOT PX_WorkArea[Mission^.PPlace] THEN // Se non vede la fotocellula, disattiva la piazzola e la dichiara libera per evitare di andare a far dei danni successivi
								WorkAreaState^[Mission^.PPlace].State := WORKAREA_STATE_FREE_DISABLED;
								Errore := ErrPALLETNOTPRESENT;
								EXIT;
							END_IF
						ELSE		//riferito al case WorkAreaManager^.State
							;
						END_CASE	//riferito al case WorkAreaManager^.State
				ELSE
					(* Controllo della Ph di presenza pallet, in base a quello gestisco lo stato della piazzola *)
					IF PX_WorkArea[cwa] THEN
						WorkAreaState^[cwa].State := WORKAREA_STATE_OCCUPIED_DISABLED;
					ELSE
						WorkAreaState^[cwa].State := WORKAREA_STATE_FREE_DISABLED;
					END_IF
				END_IF
(**********************************************************************************************************************************************************************************)
(**********************************************************************************************************************************************************************************)
			(* Occupied + Working (Gestione PACCHI/FALDE) *)
(**********************************************************************************************************************************************************************************)
(**********************************************************************************************************************************************************************************)
			WORKAREA_STATE_OCCUPIED_WORKING:
				IF WorkArea^[cwa].Enable = 1 AND Forming^[WorkAreaState^[cwa].F].Enable = 1 OR
					WorkArea^[cwa].Typology <> TYPOLOGY_PALLET OR
					((WorkArea^[cwa].Enable = 0 OR Forming^[WorkAreaState^[cwa].F].Enable = 0) AND Mission^.State > MISSION_STATE_NOP) THEN
					CASE  WorkAreaManager^.State OF
												
						WAMANAGER_NOP:
							(* Forzatura Piazzola da Estrarre. Si passa per il Tape *) 
							IF WorkArea^[cwa].LGV_Req = 1 THEN
								WorkAreaState^[cwa].State := WORKAREA_STATE_OCCUPIED_WORKED;
								RestoreCWA^ := TRUE;
								PreviousPWA^ :=cwa;
								EXIT;
							END_IF
							IF WorkAreaState^[cwa].L = 0 THEN		// se è necessario depositare la falda
								IF WorkAreaState^[cwa].P = 0 THEN 	// se non ho pacchi depositati
									(* Falda Iniziale *)
									IF Forming^[WorkAreaState^[cwa].F].Layer > 0 THEN	// se è necessario depositare ho un tipo (1..n) di falda
										(* Cerco disponibilità Falda *)
										ppick := TFPalletizerGetWAFromTypeCode(WorkArea,WorkAreaState,TYPOLOGY_LAYER,Forming^[WorkAreaState^[cwa].F].Layer);
										IF ppick > 0 AND 			// se esiste una piazzola adibita a magazzino con codice falda designato
											PX_WorkArea[ppick] THEN	// se la Fotocelula mi indica la presenza effettiva di almeno una falda
											WorkAreaManager^.State  := WAMANAGER_CICLO_FALDA_INIT;	// setto lo stato del WAMANAGER
											RestoreCWA^ := TRUE;
											PreviousPWA^ := pwa;
											EXIT;
										END_IF
									ELSE
										(* Nessuna Falda da gestire dopo Pallet/Prima del primo pacco. Assegno WorkArea^[cwa].L=1 come se fosse dopositato *)
										(* Assegno WorkArea^[cwa].P=1 per gestione primo PACCO *)
										WorkAreaState^[cwa].L := 1;
										WorkAreaState^[cwa].P := 1;
										EXIT;
									END_IF
								ELSE
									(* Falde Successive *)
									(* Cerco disponibilità Falda *)
									ppick := TFPalletizerGetWAFromTypeCode(WorkArea:=WorkArea,WorkAreaState:=WorkAreaState,Typology:=TYPOLOGY_LAYER,TCode:=Forming^[WorkAreaState^[cwa].F].PackXP[WorkAreaState^[cwa].P].Layer);
									IF ppick > 0 AND 				// se esiste una piazzola adibita a magazzino con codice falda designato
										PX_WorkArea[ppick] THEN		// se la Fotocelula mi indica la presenza effettiva di almeno una falda
										WorkAreaManager^.State  := WAMANAGER_CICLO_FALDA_INIT;	// setto lo stato del WAMANAGER
										RestoreCWA^ := TRUE;
										PreviousPWA^ := pwa;
										EXIT;
									ELSif ppick = -1 THEN
										Errore:=ErrLAYERCODENOTFOUND;
										EXIT;
									END_IF
								END_IF
							ELSE	// se non devo depositare la falda
								
								(* Assegnazione del codice con la modalità ad approccio diretto, cioè:
									- I pallet sono già stati depositati sulla WA
									- Alla WA viene assegnato il codice del pacco presente sul ribaltino solo se non è già presente una WA in lavorazione con lo stesso codice
									- Il codice assegnato alla WA rientra nei codici stabiliti dalla gestione a Zone
									- Il codice sul ribaltino è presente nella formatura attiva della WA*)	
								ppick := 1;//TFPalletizerGetWPPFromPackCode(WorkPickPointState,WorkArea^[cwa].Code);
								WAconCodiceWPPPresente := TFWAconCodiceWPPPresente(WorkArea,WorkAreaState,WorkPickPointState,ppick); // Valuto se è già presente una WA in lavorazione con il codice del pacco sul ribaltino	
								pcode := TFPackCodePresenteInZona(WorkPickPointState:=WorkPickPointState,WorkAreaZone:=WorkAreaZone,WorkArea:=cwa);//TFPackCodePresentToZone(HandlingPackTable,WorkAreaZone,cwa);
(**********************)	//	CodiceValidoPerWA := TFCodicePaccoPresenteInFormatura(Forming := Forming,IndiceFormatura := WorkAreaState^[cwa].F,CodiceInValutazione := pcode);	
								IF pcode<>0 THEN
									IF NOT TFCodicePaccoPresenteInFormaturaAll(Forming := Forming,CodiceInValutazione := pcode) THEN
										Errore:= ErrPACKCODENOTFOUND;
									END_IF
								END_IF
								IF NOT TFCodicePaccoPresenteInFormatura(Forming := Forming,IndiceFormatura := WorkAreaState^[cwa].F,CodiceInValutazione := pcode) THEN
									CodiceValidoPerWA := FALSE;
									IF pcode<>0 THEN
										;//Errore:= ErrPACKCODENOTFOUND;
									END_IF
								ELSE
									CodiceValidoPerWA := TRUE;
								END_IF
								IF WorkAreaState^[cwa].P = 1 AND WorkArea^[cwa].Initialize AND
									WorkArea^[cwa].Code = 0 AND NOT WAconCodiceWPPPresente AND 
									pcode = WorkPickPointState^[1].Code AND CodiceValidoPerWA THEN
									
									IF (ppick > 0 AND HandlingRun) AND // c'è un pacco sul ribaltino e i traspporti sono in automatico
										NOT WAconCodiceWPPPresente  AND // non è già presente una WA in lavorazione con il codice del pacco sul ribaltino
										pcode = WorkPickPointState^[ppick].Code  THEN // il codice sul ribaltino può essere assegnato alla WA in base alla suddivisione delle zone
											WorkArea^[cwa].Code := pcode;
											WorkArea^[cwa].Initialize := FALSE;
											RestoreCWA^ := TRUE;
											PreviousPWA^ := pwa;
											EXIT;
									ELSE
										EXIT;
									END_IF
								ELSE (* Cerco Disponibilità Pacco *)
									ppick := TFPalletizerGetWPPFromPackCode(WorkPickPointState,WorkArea^[cwa].Code); // Valuta se c'è un PickPoint con il pacco col codice della WA 
									ConsentiDepositoPaccoSuWA := TFConsentiDepositoPaccoSuWA(WorkArea,WorkAreaState,cwa); // Valutazione se è possibile depositare il pacco sulla WA, valuta se ci sono altre WA con il codice della WA in esame e con un numero di pacchi maggiore
			(**********************)	//	CodiceValidoPerWA := TFCodicePaccoPresenteInFormatura(Forming := Forming,IndiceFormatura := WorkAreaState^[cwa].F,CodiceInValutazione := pcode);	
										IF pcode<>0 THEN
											IF NOT TFCodicePaccoPresenteInFormaturaAll(Forming := Forming,CodiceInValutazione := pcode) THEN
												Errore:= ErrPACKCODENOTFOUND;
											END_IF
										END_IF
										IF NOT TFCodicePaccoPresenteInFormatura(Forming := Forming,IndiceFormatura := WorkAreaState^[cwa].F,CodiceInValutazione := pcode) THEN
											CodiceValidoPerWA := FALSE;
											IF pcode<>0 THEN
												;//Errore:= ErrPACKCODENOTFOUND;
											END_IF
										ELSE
											CodiceValidoPerWA := TRUE;
										END_IF
										IF (ppick > 0 AND Forming^[WorkAreaState^[cwa].F].Enable = 1) AND CodiceValidoPerWA AND ((ConsentiDepositoPaccoSuWA AND AbilitaDisposizionePalletContinua^) OR NOT AbilitaDisposizionePalletContinua^) THEN // se c'è un pacco e i trasporti (quindi il ribaltino )sono in automatico
										(* Se il grip = -1 metto la Workarea nello stato WORKAREA_STATE_OCCUPIED_WORKED*)
										IF Forming^[WorkAreaState^[cwa].F].PackXP[WorkAreaState^[cwa].P].Grip = -1 OR
											Forming^[WorkAreaState^[cwa].F].PackXN[WorkAreaState^[cwa].P].Grip = -1 THEN
											WorkAreaState^[cwa].State := WORKAREA_STATE_OCCUPIED_WORKED;
											WorkAreaManager^.State  := WAMANAGER_NOP;
											CicloDiRiposoNecessario := TRUE;
											EXIT;
										ELSE
											(* Aggiorno l'Array dei Codici Usati *)
											//TFRefreshUsedCode(WorkArea^[cwa].Code,UsedCode);
											IF (AbilitaComandiAnticipatiRibaltino AND HandlingOKPrelievoPacco) OR 	// Se c'è l'abilitazione degli antici del ribaltino e il ribaltino è in condizioni di dare il pacco
												(NOT AbilitaComandiAnticipatiRibaltino AND HandlingRun) THEN		// Se NON c'è l'abilitazione dei comandi anticipati del ribaltino e i trasporti sono in automatico
												WorkAreaManager^.State  := WAMANAGER_CICLO_PACCO_INIT;				// Setto lo stato del WAMANAGER
												RestoreCWA^ := TRUE;
												PreviousPWA^ := pwa;
												UltimaWAAssegnazionePacco := cwa;
												CicloDiRiposoNecessario := FALSE;
												EXIT;
											END_IF
										END_IF
									ELSE
										IF Forming^[WorkAreaState^[cwa].F].Enable = 1 THEN
											(* Se il grip = -1 metto la Workarea nello stato WORKAREA_STATE_OCCUPIED_WORKED*)
											IF Forming^[WorkAreaState^[cwa].F].PackXP[WorkAreaState^[cwa].P].Grip = -1 OR
												Forming^[WorkAreaState^[cwa].F].PackXN[WorkAreaState^[cwa].P].Grip = -1 THEN
												WorkAreaState^[cwa].State := WORKAREA_STATE_OCCUPIED_WORKED;
												WorkAreaManager^.State  := WAMANAGER_NOP;
												EXIT;
											END_IF
										END_IF
										;//CicloDiRiposoNecessario := TRUE;
									END_IF
								END_IF
							END_IF
								
							
						WAMANAGER_CICLO_FALDA_INIT:
							
							(* Creo Missione Falda *)
							Mission^.PPick			:= ppick; 				// valorizzo il punto di prelievo = workarea dove ho valutato la presenza delle falde
							Mission^.TPick 			:= TPICK_LAYER;			// valorizzo la tipologia di prelievo = tipo prelievo falda
							Mission^.PPlace			:= cwa;					// valorizzo il punto di deposito = workarea dove ho valutato di depositare la falda
							Mission^.XPick			:= WorkArea^[Mission^.PPick].X + WorkAreaOffset^[Mission^.PPick].X;// + (Layer^[WorkArea^[Mission^.PPick].Layer].X / 2); // valorizzo la quota X di prelievo 
							CASE TIPO_MAGAZZINO_FALDE OF
								MAGAZZINO_FALDE_CENTRO_FISSO:
									Mission^.YPick			:= WorkArea^[Mission^.PPick].Y + WorkAreaOffset^[Mission^.PPick].Y;// + (Layer^[WorkArea^[Mission^.PPick].Layer].Y / 2);
								MAGAZZINO_FALDE_CENTRO_VARIABILE:
									Mission^.YPick			:= WorkArea^[Mission^.PPick].Y + WorkAreaOffset^[Mission^.PPick].Y + (Layer^[WorkArea^[Mission^.PPick].Layer].Y / 2);
							END_CASE
							
							//IF  WorkArea^[Mission^.PPick].DoLearn_Z = 1 THEN // se devo eseguire l'apprendimento della quota Z vado alla quota preposta di Start lenta
							//	Mission^.ZPick	:= WorkArea^[Mission^.PPick].Learn_Z; (* Quota di inizio apprendimento *)
							//ELSE
							//	Mission^.ZPick	:= WorkArea^[Mission^.PPick].Z + WorkArea^[Mission^.PPick].H; (* Posizione WorkArea + Altezza Reale *)
							//END_IF
							
							//IF  WorkArea^[Mission^.PPick].DoLearn_Z = 1 THEN 	// se devo fare l'apprendimento sulla catasta vuoti
								Mission^.ZPick	:= WorkArea^[Mission^.PPick].Z; // in questo modo LA LENTA va sempre fino a zero...mi fermo al raggiungimento dell'intervento dei tastatori
							//ELSE											// se NON devo fare l'apprendimento sulla catasta vuoti
							//	Mission^.ZPick		:= WorkArea^[Mission^.PPick].Z + WorkArea^[Mission^.PPick].H; //quota reale catasta vuoti = (altezza WA + altezza reale)
							//END_IF
					
